IF st_config.b_config_fertig THEN
	(* Fehlermeldungen und Betriebsmeldungen ab dem Startindex in die globalen Meldungsarrays schreiben *)
	garr_stoermeldungen[st_config.i16_meld_startindex + 0] := sm_haspel_notaus;
	garr_stoermeldungen[st_config.i16_meld_startindex + 1] := sm_haspel_notabschaltung;
	garr_stoermeldungen[st_config.i16_meld_startindex + 2] := FALSE;
	garr_stoermeldungen[st_config.i16_meld_startindex + 3] := FALSE;
	garr_stoermeldungen[st_config.i16_meld_startindex + 4] := FALSE;
	garr_stoermeldungen[st_config.i16_meld_startindex + 5] := FALSE;
	garr_stoermeldungen[st_config.i16_meld_startindex + 6] := FALSE;
	garr_stoermeldungen[st_config.i16_meld_startindex + 7] := FALSE;
	garr_stoermeldungen[st_config.i16_meld_startindex + 8] := FALSE;
	garr_stoermeldungen[st_config.i16_meld_startindex + 9] := FALSE;
	garr_stoermeldungen[st_config.i16_meld_startindex + 10] := FALSE;
	garr_stoermeldungen[st_config.i16_meld_startindex + 11] := FALSE;
	garr_stoermeldungen[st_config.i16_meld_startindex + 12] := FALSE;
	garr_stoermeldungen[st_config.i16_meld_startindex + 13] := FALSE;
	garr_stoermeldungen[st_config.i16_meld_startindex + 14] := FALSE;
	garr_stoermeldungen[st_config.i16_meld_startindex + 15] := FALSE;
	garr_stoermeldungen[st_config.i16_meld_startindex + 16] := FALSE;
	garr_stoermeldungen[st_config.i16_meld_startindex + 17] := FALSE;
	garr_stoermeldungen[st_config.i16_meld_startindex + 18] := FALSE;
	garr_stoermeldungen[st_config.i16_meld_startindex + 19] := FALSE;
	
	garr_betriebsmeldungen[st_config.i16_meld_startindex + 0] := bm_haspel_bandende;
	garr_betriebsmeldungen[st_config.i16_meld_startindex + 1] := FALSE;
	garr_betriebsmeldungen[st_config.i16_meld_startindex + 2] := FALSE;
	garr_betriebsmeldungen[st_config.i16_meld_startindex + 3] := FALSE;
	garr_betriebsmeldungen[st_config.i16_meld_startindex + 4] := FALSE;
	garr_betriebsmeldungen[st_config.i16_meld_startindex + 5] := FALSE;
	garr_betriebsmeldungen[st_config.i16_meld_startindex + 6] := FALSE;
	garr_betriebsmeldungen[st_config.i16_meld_startindex + 7] := FALSE;
	garr_betriebsmeldungen[st_config.i16_meld_startindex + 8] := FALSE;
	garr_betriebsmeldungen[st_config.i16_meld_startindex + 9] := FALSE;
	garr_betriebsmeldungen[st_config.i16_meld_startindex + 10] := FALSE;
	garr_betriebsmeldungen[st_config.i16_meld_startindex + 11] := FALSE;
	garr_betriebsmeldungen[st_config.i16_meld_startindex + 12] := FALSE;
	garr_betriebsmeldungen[st_config.i16_meld_startindex + 13] := FALSE;
	garr_betriebsmeldungen[st_config.i16_meld_startindex + 14] := FALSE;
	garr_betriebsmeldungen[st_config.i16_meld_startindex + 15] := FALSE;
	garr_betriebsmeldungen[st_config.i16_meld_startindex + 16] := FALSE;
	garr_betriebsmeldungen[st_config.i16_meld_startindex + 17] := FALSE;
	garr_betriebsmeldungen[st_config.i16_meld_startindex + 18] := FALSE;
	garr_betriebsmeldungen[st_config.i16_meld_startindex + 19] := FALSE;
END_IF
END_FUNCTION_BLOCK

(* POU EPT Lib/CamEditor/ST_Kurvenscheibeneditor, ST *)
FUNCTION_BLOCK ST_Kurvenscheibeneditor
VAR_INPUT
 	udint_camtable_id						: UDINT;
	i16_laenge_mfp_tabelle				: UINT;
	arr_db_mfps							: ARRAY[1..ui_MAX_NUM_MFP] OF struct_db_motionfunctionpoint;	(* Vorgabe aus der Datenbank *)
	st_config								: struct_config;
	st_ctrl_in								: struct_ctrl_in;
END_VAR
VAR_IN_OUT
	i16_auftrag							: enum_auftrag_cameditor;
END_VAR
VAR_OUTPUT
	st_ctrl_out							: struct_ctrl_out;
END_VAR
VAR
	mc_point_id							: MC_MotionFunctionPoint_ID;
	mc_read_motion_function_point			: MC_ReadMotionFunctionPoint;
	mc_write_motion_function_point			: MC_WriteMotionFunctionPoint;
	arr_motion_function_points				: ARRAY[1..ui_MAX_NUM_MFP] OF MC_MotionFunctionPoint;	(* Eingelesene Kurvenscheibentabelle aus dem Systemmanager oder geschriebene MFPs an den Systemmanager *)
	udint_write_error_id 					: UDINT := 0;
	udint_read_error_id					: UDINT := 0;
	fb_state_entry							: ST_StateEntry;
	fb_ton_quitt							: TON;
	fb_ton_wz							: TON;
	fb_r_trig_ibn_lesen					: R_TRIG;
	fb_r_trig_ibn_schreiben					: R_TRIG;
	fb_ton_ibn_lesen						: TON;
	fb_ton_ibn_schreiben					: TON;
	b_ibn_lesen							: BOOL := FALSE;
	b_ibn_schreiben						: BOOL := FALSE;
	sm_fehler_schreibe_mfp 				: BOOL := FALSE;
	sm_fehler_lese_mfp					: BOOL := FALSE;
END_VAR
VAR CONSTANT
	ui_MAX_NUM_MFP					:UINT := 100;
END_VAR
fb_ton_wz(IN:= , PT:= , Q=> , ET=> );
fb_ton_quitt(IN:= , PT:= t#100ms, Q=> , ET=> );

fb_r_trig_ibn_lesen(CLK:= b_ibn_lesen, Q=> );
fb_r_trig_ibn_schreiben(CLK:= b_ibn_schreiben, Q=> );
fb_ton_ibn_lesen(IN:= , PT:= t#1s, Q=> , ET=> );
fb_ton_ibn_schreiben(IN:= , PT:= t#1s, Q=> , ET=> );


IF fb_r_trig_ibn_lesen.Q THEN
	fb_ton_ibn_lesen.IN := TRUE;
ELSE
	IF fb_ton_ibn_lesen.Q THEN
		b_ibn_lesen := FALSE;
	 	fb_ton_ibn_lesen.IN := FALSE;
	END_IF
END_IF

IF fb_r_trig_ibn_schreiben.Q THEN
	fb_ton_ibn_schreiben.IN := TRUE;
ELSE
	IF fb_ton_ibn_schreiben.Q THEN
		b_ibn_schreiben := FALSE;
	 	fb_ton_ibn_schreiben.IN := FALSE;
	END_IF
END_IF

(* ======================================Schrittkette======================================== *)
fb_state_entry(
	i16_next_step:= ,
	i16_pos:= 1,
	s_debugtext:= ,
	E=> ,
	X=> ,
	i16_step=> ,
	i16_last_step=> );

CASE fb_state_entry.i16_step OF
(*=======================================================*)
	0:	(* Init *)
		fb_ton_quitt.IN := FALSE;
		st_ctrl_out.b_bereit := FALSE;
		st_ctrl_out.b_fehler := FALSE;
		i16_auftrag := MFP_KEIN_AUFTRAG;
		mc_point_id := 1;
		mc_read_motion_function_point.Execute := FALSE;
		mc_write_motion_function_point.Execute := FALSE;
		sm_fehler_schreibe_mfp := FALSE;
		sm_fehler_lese_mfp := FALSE;
		fb_state_entry.i16_next_step := 10;

(*=======================================================*)
	10: (* Warte auf Auftrag *)
		IF fb_state_entry.E THEN
			st_ctrl_out.b_bereit := TRUE;
		END_IF

		(* Motion Function Points aus der Kurvenscheibentabelle des Systemmanagers lesen *)
		IF i16_auftrag = MFP_LESEN OR fb_r_trig_ibn_lesen.Q THEN
			fb_state_entry.i16_next_step := 100;
		(* Motion Function Points von der Datenbankvorgabe in die Kurvenscheibentabelle des Systemmanagers schreiben *)
		ELSIF i16_auftrag = MFP_SCHREIBEN OR fb_r_trig_ibn_schreiben.Q THEN
			fb_state_entry.i16_next_step := 200;
		END_IF

(*=======================================================*)
	100:
		mc_point_id := 1;
		fb_state_entry.i16_next_step := 110;

(*=======================================================*)
	110:	(* Lese die einzelnen MFPs aus der Kurvenscheibentabelle des Systemmanagers *)
		IF fb_state_entry.E THEN
			mc_read_motion_function_point.Execute := TRUE;
		END_IF

		IF mc_read_motion_function_point.Busy THEN
			mc_read_motion_function_point.Execute := FALSE;
			fb_state_entry.i16_next_step := 120;
		END_IF

(*=======================================================*)
	120:	(* MFP wurde gelesen *)
		IF  NOT mc_read_motion_function_point.Busy THEN
			IF NOT mc_read_motion_function_point.Error THEN
				fb_state_entry.i16_next_step := 130;
			ELSE
				sm_fehler_schreibe_mfp := TRUE;
				fb_state_entry.i16_next_step := FEHLER;
			END_IF
		END_IF

(*=======================================================*)
	130:	(* Zum nächsten MFP *)
		IF fb_state_entry.E THEN
			mc_point_id := mc_point_id + 1;
		END_IF

		IF mc_point_id > i16_laenge_mfp_tabelle THEN
			(* Alle Punkte wurden gelesen *)
			fb_state_entry.i16_next_step := 140;
		ELSE
			(* Weitere Punkte lesen *)
			fb_state_entry.i16_next_step := 110;
		END_IF

(*=======================================================*)
	140:	(* Lesevorgang beendet *)
		fb_state_entry.i16_next_step := 0;

(*=======================================================*)
	200:	(* Einlesen der Vorgabepunktetabelle *)
		IF fb_state_entry.E THEN
			FOR mc_point_id := 1  TO 32 BY 1DO
				arr_motion_function_points[mc_point_id].PointIndex := arr_db_mfps[mc_point_id].PointIndex;
				arr_motion_function_points[mc_point_id].FunctionType := arr_db_mfps[mc_point_id].FunctionType;
				arr_motion_function_points[mc_point_id].PointType := arr_db_mfps[mc_point_id].PointType;
				arr_motion_function_points[mc_point_id].RelIndexNextPoint := 1;
				arr_motion_function_points[mc_point_id].MasterPos := arr_db_mfps[mc_point_id].MasterPos;
				arr_motion_function_points[mc_point_id].SlavePos := arr_db_mfps[mc_point_id].SlavePos;
			END_FOR
		END_IF
		mc_point_id := 1;
		fb_state_entry.i16_next_step := 210;

(*=======================================================*)
	210:	(* Schreibe die einzelnen MFPs *)
		IF fb_state_entry.E THEN
			mc_write_motion_function_point.Execute := TRUE;
		END_IF

		IF mc_write_motion_function_point.Busy THEN
			mc_write_motion_function_point.Execute := FALSE;
			fb_state_entry.i16_next_step := 220;
		END_IF

(*=======================================================*)
	220:	(* MFP wurde geschrieben *)
		IF  NOT mc_write_motion_function_point.Busy THEN
			IF NOT  mc_write_motion_function_point.Error THEN
				fb_state_entry.i16_next_step := 230;
			ELSE
				sm_fehler_schreibe_mfp := TRUE;
				fb_state_entry.i16_next_step := FEHLER;
			END_IF
		END_IF

(*=======================================================*)
	230:	(* Zum nächsten MFP *)
		IF fb_state_entry.E THEN
			mc_point_id := mc_point_id + 1;
		END_IF

		IF mc_point_id > i16_laenge_mfp_tabelle THEN
			(* Alle Punkte wurden gelesen *)
			fb_state_entry.i16_next_step := 240;
		ELSE
			(* Weitere Punkte lesen *)
			fb_state_entry.i16_next_step := 210;
		END_IF

(*=======================================================*)
	240:	(* Schreibevorgang beendet *)
		fb_state_entry.i16_next_step := 0;

(*=======================================================*)
	1000: (* Fehler *)
		IF fb_state_entry.E THEN
			st_ctrl_out.b_fehler := TRUE;
			fb_ton_quitt.IN := FALSE;
		END_IF

		(*-----------------------Weiterschaltbedingungen----------------------------*)
		IF st_ctrl_in.b_quitt AND NOT fb_state_entry.E THEN
			st_ctrl_out.b_fehler := FALSE;
			fb_ton_quitt.IN := TRUE;
		END_IF

		IF fb_ton_quitt.Q THEN
			fb_ton_quitt.IN := FALSE;
			fb_state_entry.i16_next_step := 0;
		END_IF
END_CASE

fb_state_entry(
	i16_next_step:= ,
	i16_pos:= 2,
	s_debugtext:= ,
	E=> ,
	X=> ,
	i16_step=> ,
	i16_last_step=> );

mc_read_motion_function_point(
	Execute:= ,
	CamTableID:= udint_camtable_id,
	PointID:= mc_point_id,
	Point:= arr_motion_function_points[mc_point_id],
	Done=> , 
	Busy=> , 
	Error=> , 
	ErrorID=> );

mc_write_motion_function_point(
	Execute:= , 
	CamTableID:= udint_camtable_id,
	PointID:= mc_point_id,
	Point:= arr_motion_function_points[mc_point_id],
	Done=> , 
	Busy=> , 
	Error=> , 
	ErrorID=> );

IF st_config.b_config_fertig THEN
	garr_stoermeldungen[st_config.i16_meld_startindex + 0] := sm_fehler_lese_mfp;
	garr_stoermeldungen[st_config.i16_meld_startindex + 1] := sm_fehler_schreibe_mfp;
	garr_stoermeldungen[st_config.i16_meld_startindex + 2] := FALSE;
	garr_stoermeldungen[st_config.i16_meld_startindex + 3] := FALSE;
	garr_stoermeldungen[st_config.i16_meld_startindex + 4] := FALSE;
	garr_stoermeldungen[st_config.i16_meld_startindex + 5] := FALSE;
	garr_stoermeldungen[st_config.i16_meld_startindex + 6] := FALSE;
	garr_stoermeldungen[st_config.i16_meld_startindex + 7] := FALSE;
	garr_stoermeldungen[st_config.i16_meld_startindex + 8] := FALSE;
	garr_stoermeldungen[st_config.i16_meld_startindex + 9] := FALSE;
	garr_stoermeldungen[st_config.i16_meld_startindex + 10] := FALSE;
	garr_stoermeldungen[st_config.i16_meld_startindex + 11] := FALSE;
	garr_stoermeldungen[st_config.i16_meld_startindex + 12] := FALSE;
	garr_stoermeldungen[st_config.i16_meld_startindex + 13] := FALSE;
	garr_stoermeldungen[st_config.i16_meld_startindex + 14] := FALSE;
	garr_stoermeldungen[st_config.i16_meld_startindex + 15] := FALSE;
	garr_stoermeldungen[st_config.i16_meld_startindex + 16] := FALSE;
	garr_stoermeldungen[st_config.i16_meld_startindex + 17] := FALSE;
	garr_stoermeldungen[st_config.i16_meld_startindex + 18] := FALSE;
	garr_stoermeldungen[st_config.i16_meld_startindex + 19] := FALSE;
	
	garr_betriebsmeldungen[st_config.i16_meld_startindex + 0] := FALSE;
	garr_betriebsmeldungen[st_config.i16_meld_startindex + 1] := FALSE;
	garr_betriebsmeldungen[st_config.i16_meld_startindex + 2] := FALSE;
	garr_betriebsmeldungen[st_config.i16_meld_startindex + 3] := FALSE;
	garr_betriebsmeldungen[st_config.i16_meld_startindex + 4] := FALSE;
	garr_betriebsmeldungen[st_config.i16_meld_startindex + 5] := FALSE;
	garr_betriebsmeldungen[st_config.i16_meld_startindex + 6] := FALSE;
	garr_betriebsmeldungen[st_config.i16_meld_startindex + 7] := FALSE;
	garr_betriebsmeldungen[st_config.i16_meld_startindex + 8] := FALSE;
	garr_betriebsmeldungen[st_config.i16_meld_startindex + 9] := FALSE;
	garr_betriebsmeldungen[st_config.i16_meld_startindex + 10] := FALSE;
	garr_betriebsmeldungen[st_config.i16_meld_startindex + 11] := FALSE;
	garr_betriebsmeldungen[st_config.i16_meld_startindex + 12] := FALSE;
	garr_betriebsmeldungen[st_config.i16_meld_startindex + 13] := FALSE;
	garr_betriebsmeldungen[st_config.i16_meld_startindex + 14] := FALSE;
	garr_betriebsmeldungen[st_config.i16_meld_startindex + 15] := FALSE;
	garr_betriebsmeldungen[st_config.i16_meld_startindex + 16] := FALSE;
	garr_betriebsmeldungen[st_config.i16_meld_startindex + 17] := FALSE;
	garr_betriebsmeldungen[st_config.i16_meld_startindex + 18] := FALSE;
	garr_betriebsmeldungen[st_config.i16_meld_startindex + 19] := FALSE;
END_IF
END_FUNCTION_BLOCK

(* POU EPT Lib/CamEditor/Verfahrberechnungen/ST_MFCalcConstPhase, ST *)
FUNCTION_BLOCK ST_MFCalcConstPhase
VAR_INPUT
	st_config								: struct_config;
	st_ctrl_in								: struct_ctrl_in;

	(* Kurvenscheibendaten *)
	udiTableId							: MC_CAM_ID;			(* Table-ID *)
	eMotionFunctionType					: MC_MotionFunctionType;	(*Bewegungsgesetz: MOTIONFUNCTYPE_POLYNOM5 etc.*)
	i16_startpunkt_edit_mf_tab				: INT;
	arr_db_mf_tab						: ARRAY[1..i_MAX_NUM_MFP] OF struct_db_motionfunctionpoint;	(* Vorgabe aus der Datenbank *)

	(* Bewegungsdaten an der Last *)
	lrVeloMax							: LREAL;	(*maximale Geschwindigkeit [mm/s] an der Last *)
	lrAccMax								: LREAL;	(*maximale Beschleunigung [mm/s²] an der Last *)
	lrDecMax							: LREAL;	(*maximale Beschleunigung [mm/s²] an der Last *)

	lrModuloValue 						: LREAL ;
END_VAR
VAR_IN_OUT
	st_AxisRefMaster						: AXIS_REF;
	st_AxisRefSlave						: AXIS_REF;
END_VAR
VAR_OUTPUT
	lrMasterVeloMax						: LREAL;	(* Maximum Master Velocity [°/s] *)
	lrMasterRotPerMinMax					: LREAL;	(* Maximum Master Rotations per Minute [1/min] *)
	st_ctrl_out							: struct_ctrl_out;
END_VAR
VAR
	st_sm						 		: struct_cameditor_meldungen;
	fb_state_entry							: ST_StateEntry;
	fb_ton_quitt							: TON;
	fb_ton_wz							: TON;

	stMotionFunctionPointDummy			: MC_MotionFunctionPoint;	(* Dummy-Punkt *)
(*	TYPE MC_MotionFunctionPoint :
		STRUCT
		    PointIndex        		: MC_MotionFunctionPoint_ID;
		    FunctionType   		: MC_MotionFunctionType;
		    PointType         		: MC_MotionPointType;
		    RelIndexNextPoint 	: MC_MotionFunctionPoint_ID;
		    MasterPos         		: LREAL; (* X *)
		    SlavePos          		: LREAL; (* Y *)
		    SlaveVelo         		: LREAL; (* Y' *)
		    SlaveAcc          		: LREAL; (* Y'' *)
		    SlaveJerk         		: LREAL; (* Y''' *)
		END_STRUCT
	END_TYPE
*)

	(*Motion Function runterschreiben an NC*)
	astWriteMotionFunction 				: ARRAY[1..i_MAX_NUM_MFP] OF MC_MotionFunctionPoint;
	stWriteMFCamTableRef				: MC_CAM_Ref;	(*Definition Zieltabelle*)
	fbCamTableSelect					: MC_CamTableSelect;
	fbWriteMF							: MC_WriteMotionFunction;
	b_cam_table_select_periodic			: BOOL := FALSE;
	b_cam_table_select_master_absolute	: BOOL := FALSE;
	b_cam_table_select_slave_absolute		: BOOL := FALSE;

	(*Motion Function hochladen von NC*)
	fbReadMF							: MC_ReadMotionFunction;
	stReadMFCamTableRef				: MC_CAM_Ref;	(*Definition Zieltabelle*)
	astReadMotionFunction 				: ARRAY[0..i_MAX_NUM_MFP] OF MC_MotionFunctionPoint;

	(*Berechnung Konstantfahrphase*)
	fbMFcalcConstVelo					: ST_MFcalcConstVelo;	(*Baustein zur Berechnung, ob eine Konstantfahphase möglich ist*)
	stDataCalcConstVelo 					: ARRAY[1..4] OF MC_MotionFunctionPoint;	(*Aus der Berechnung ermittelte Punktedaten*)

	(* Berechnung Mastergeschwindigkeit*)
	fbMFMaxMasterVelo					: ST_MFMaxMasterVelo;	(* Baustein zur Berechnung der maximalen Mastergeschwindigkeit *)

	(*Temporäre Variablen *)
	iPointCount							: INT := 0;
	iNumMfPoints							: INT := 0;
	i_point_nr							: INT := 0;
	err_id								: UDINT := 0;
	i16_anzahl_mfps						: INT;
	lrStartPointMaster						: LREAL;	(* Startpunkt Master [°] *)
	lrStartPointSlave						: LREAL;	(* Startpunkt Slave [mm] *)
	lrEndPointMaster						: LREAL;	(* Endpunkt Master [°] *)
	lrEndPointSlave						: LREAL;	(* Endpunkt Slave [mm] *)
	lr_anfang_cam_table					: LREAL := 0;	(* Anfang Darstellungsbereich MF-Tabelle *)
	lr_ende_cam_table					: LREAL := 0;	(* Ende Darstellungsbereich MF-Tabelle *)
END_VAR
VAR CONSTANT
	i_MAX_NUM_MFP						: INT := 100;
END_VAR
fb_ton_wz(IN:= , PT:= , Q=> , ET=> );
fb_ton_quitt(IN:= , PT:= t#50ms, Q=> , ET=> );

(* ======================================Schrittkette======================================== *)
fb_state_entry(
	i16_next_step:= ,
	i16_pos:= 1,
	s_debugtext:= ,
	E=> ,
	X=> ,
	i16_step=> ,
	i16_last_step=> );

CASE fb_state_entry.i16_step OF
(*=======================================================*)
	0:	(* Init *)
		st_ctrl_out.b_bereit := FALSE;
		st_ctrl_out.b_fertig := FALSE;
		st_ctrl_out.b_fehler := FALSE;
		fbCamTableSelect.Execute := FALSE;
		fbWriteMF.Execute := FALSE;
		fbReadMF.Execute := FALSE;
		fbMFMaxMasterVelo.bExecute := FALSE;
		fbMFcalcConstVelo.bExecute := FALSE;
		err_id := 0;
		i16_anzahl_mfps := 0;
		st_sm.berechne_konstantfahrphase := FALSE;
		st_sm.berechne_max_master_geschwindigkeit := FALSE;
		st_sm.lese_camtable := FALSE;
		st_sm.lese_mfp := FALSE;
		st_sm.lesen_werte_mf_tab := FALSE;
		st_sm.schreibe_camtable := FALSE;
		st_sm.schreibe_mfp := FALSE;

		fb_state_entry.i16_next_step := 10;

(*=======================================================*)
	10:	(* Warte auf Start *)
		IF lrModuloValue > 0 THEN
			b_cam_table_select_periodic := TRUE;
			b_cam_table_select_master_absolute := TRUE;
			b_cam_table_select_slave_absolute := FALSE;
		ELSE
			b_cam_table_select_periodic := FALSE;
			b_cam_table_select_master_absolute := TRUE;
			b_cam_table_select_slave_absolute := TRUE;
		END_IF

		(*-----------------------Weiterschaltbedingungen----------------------------*)
		IF st_ctrl_in.b_start THEN
			i16_anzahl_mfps := 0;
			lrMasterVeloMax := 0;
			lrMasterRotPerMinMax := 0;
			fb_state_entry.i16_next_step := 100;
		END_IF

(*=======================================================*)
	100:	(*  *)
		IF fb_state_entry.E THEN
			FOR i_point_nr := 1 TO i_MAX_NUM_MFP BY 1 DO
				(*Für Download: Initialisieren aller  MFPs im Array *)
				astWriteMotionFunction[i_point_nr] := stMotionFunctionPointDummy;
				astWriteMotionFunction[i_point_nr].RelIndexNextPoint  := 1;

				(* Übernahme der Daten aus der WKZ-Datenbank *)
				astWriteMotionFunction[i_point_nr].FunctionType := arr_db_mf_tab[i_point_nr].FunctionType;
				astWriteMotionFunction[i_point_nr].MasterPos  := arr_db_mf_tab[i_point_nr].MasterPos;
				astWriteMotionFunction[i_point_nr].SlavePos  := arr_db_mf_tab[i_point_nr].SlavePos;
				astWriteMotionFunction[i_point_nr].PointType  := arr_db_mf_tab[i_point_nr].PointType;
				astWriteMotionFunction[i_point_nr].PointIndex  := arr_db_mf_tab[i_point_nr].PointIndex;

				IF astWriteMotionFunction[i_point_nr].FunctionType > MOTIONFUNCTYPE_NOTDEF THEN
					i16_anzahl_mfps := i16_anzahl_mfps + 1;
				END_IF
			END_FOR

			(* Beim Letzen Punkt in der Tabelle immer den RelIndexNextPoint auf 0 setzen *)
			astWriteMotionFunction[i16_anzahl_mfps].RelIndexNextPoint := 0;

			(* Darstellungsbereich der MF-Tabelle (wird benötigt für die Funktion "MC_ReadMotionFunctionValues") *)
			IF lrModuloValue > 0 THEN
				lr_anfang_cam_table := 0;
				lr_ende_cam_table := lrModuloValue;
			ELSE
				lr_anfang_cam_table := arr_db_mf_tab[1].MasterPos;
				lr_ende_cam_table := arr_db_mf_tab[i16_anzahl_mfps].MasterPos;
			END_IF
		END_IF

		(*-----------------------Weiterschaltbedingungen----------------------------*)
		fb_state_entry.i16_next_step := 110;


(*=======================================================*)
	110:	(* Starte Berechnung der Konstantfahrphase *)
		IF fb_state_entry.E THEN
			fbMFcalcConstVelo.bExecute := TRUE;
		END_IF

		(*-----------------------Weiterschaltbedingungen----------------------------*)
		IF fbMFcalcConstVelo.bBusy THEN
			fb_state_entry.i16_next_step := 120;
		END_IF

(*=======================================================*)
	120:	(* Starte Berechnung der Konstantfahrphase *)
		IF NOT fbMFcalcConstVelo.bBusy THEN
			IF fbMFcalcConstVelo.bDone THEN
				fbMFcalcConstVelo.bExecute := FALSE;
				IF fbMFcalcConstVelo.bConstantVelo THEN
					iNumMfPoints := i16_anzahl_mfps + 2;
					fb_state_entry.i16_next_step := 130;
				ELSE
					iNumMfPoints := i16_anzahl_mfps;
					fb_state_entry.i16_next_step := 140;
				END_IF
			ELSIF fbMFcalcConstVelo.bError THEN
				st_sm.berechne_konstantfahrphase := TRUE;
				fb_state_entry.i16_next_step := 1000;
			END_IF
		END_IF

(*=======================================================*)
	130:	(* Auswertung ob Konstantfahrphase *)
		IF fb_state_entry.E THEN
			(* Verschieben aller weiteren Punkte um 2 Positionen nach hinten *)
			FOR i_point_nr := iNumMfPoints TO (i16_startpunkt_edit_mf_tab + 1) BY -1 DO
				astWriteMotionFunction[i_point_nr] := astWriteMotionFunction[i_point_nr - 2];
				astWriteMotionFunction[i_point_nr].PointIndex := i_point_nr;
			END_FOR

			iPointCount := i16_startpunkt_edit_mf_tab;

			(*Startpunkt: spezifische Daten anpassen*)
			astWriteMotionFunction[iPointCount].MasterPos := stDataCalcConstVelo[1].MasterPos;
			astWriteMotionFunction[iPointCount].SlavePos := stDataCalcConstVelo[1].SlavePos;
			astWriteMotionFunction[iPointCount].SlaveVelo := stDataCalcConstVelo[1].SlaveVelo;
			astWriteMotionFunction[iPointCount].SlaveJerk := stDataCalcConstVelo[1].SlaveJerk;
			(*Punktetyp eintragen*)
			astWriteMotionFunction[iPointCount].RelIndexNextPoint := 1;
			astWriteMotionFunction[iPointCount].FunctionType := stDataCalcConstVelo[1].FunctionType;
			astWriteMotionFunction[iPointCount].PointIndex := iPointCount;
			astWriteMotionFunction[iPointCount].PointType := stDataCalcConstVelo[1].PointType;

			iPointCount := iPointCount + 1;

			(*Zwischenpunkt 1: Konstantfahrphase eintragen*)
			astWriteMotionFunction[iPointCount].MasterPos := stDataCalcConstVelo[2].MasterPos;
			astWriteMotionFunction[iPointCount].SlavePos := stDataCalcConstVelo[2].SlavePos;
			astWriteMotionFunction[iPointCount].SlaveVelo := stDataCalcConstVelo[2].SlaveVelo;
			astWriteMotionFunction[iPointCount].SlaveJerk := stDataCalcConstVelo[2].SlaveJerk;
			(*Punktetyp eintragen*)
			astWriteMotionFunction[iPointCount].RelIndexNextPoint := 1;
			astWriteMotionFunction[iPointCount].FunctionType := stDataCalcConstVelo[2].FunctionType;
			astWriteMotionFunction[iPointCount].PointIndex := iPointCount;
			astWriteMotionFunction[iPointCount].PointType := stDataCalcConstVelo[2].PointType;
	
			iPointCount := iPointCount + 1;
	
			(*Zwischenpunkt 2: Konstantfahrphase eintragen*)
			astWriteMotionFunction[iPointCount].MasterPos := stDataCalcConstVelo[3].MasterPos;
			astWriteMotionFunction[iPointCount].SlavePos := stDataCalcConstVelo[3].SlavePos;
			astWriteMotionFunction[iPointCount].SlaveVelo := stDataCalcConstVelo[3].SlaveVelo;
			astWriteMotionFunction[iPointCount].SlaveJerk := stDataCalcConstVelo[3].SlaveJerk;
			(*Punktetyp eintragen*)
			astWriteMotionFunction[iPointCount].RelIndexNextPoint := 1;
			astWriteMotionFunction[iPointCount].FunctionType := stDataCalcConstVelo[3].FunctionType;
			astWriteMotionFunction[iPointCount].PointIndex := iPointCount;
			astWriteMotionFunction[iPointCount].PointType := stDataCalcConstVelo[3].PointType;

			iPointCount := iPointCount + 1;

			(* Beim Letzen Punkt in der Tabelle immer den RelIndexNextPoint auf 0 setzen *)
			astWriteMotionFunction[i16_anzahl_mfps + 2].RelIndexNextPoint := 0;
		END_IF

		(*-----------------------Weiterschaltbedingungen----------------------------*)
		fb_state_entry.i16_next_step := 140;

(*=======================================================*)
	140:	(* Alle Punkte der MF-Tabelle werden an die NC runter geschrieben  *)
		IF fb_state_entry.E THEN
			(*Tabelle initialisieren *)
			stWriteMFCamTableRef.pArray := ADR(astWriteMotionFunction[1]);	(* Adresse des ersten eindimensionalen Arrays vom Typ MC_MotionFunctionPoint. Jedes Array-Element enthält eine Beschreibung einer Stützstelle der Kurvenscheibe. *)
			stWriteMFCamTableRef.ArraySize := SIZEOF(astWriteMotionFunction[1]) * iNumMfPoints;
			stWriteMFCamTableRef.TableType := MC_TABLETYPE_MOTIONFUNCTION;
			stWriteMFCamTableRef.NoOfColumns := 1;	(* Bei Table Type "MC_TABLETYPE_MOTIONFUNCTION" ist NoOfColumns immer 1 *)
			stWriteMFCamTableRef.NoOfRows := iNumMfPoints;

			fbCamTableSelect.Execute := TRUE;
		END_IF

		(*-----------------------Weiterschaltbedingungen----------------------------*)
		IF fbCamTableSelect.Busy THEN
			fb_state_entry.i16_next_step := 150;
		END_IF

(*=======================================================*)
	150:	(* Alle Punkte der MF-Tabelle werden an die NC runter geschrieben  *)
		IF NOT fbCamTableSelect.Busy THEN
			IF fbCamTableSelect.Done THEN
				fbCamTableSelect.Execute := FALSE;
				fb_state_entry.i16_next_step := 200;
			ELSIF fbCamTableSelect.Error THEN
				st_sm.schreibe_camtable := TRUE;
				err_id := fbCamTableSelect.ErrorID;
				fb_state_entry.i16_next_step := 1000;
			END_IF
		END_IF

(*=======================================================*)
	200:	(* Lesen der MF-Tabelle von der NC  *)
		IF fb_state_entry.E THEN
			stReadMFCamTableRef.pArray := ADR(astReadMotionFunction[0]);
			stReadMFCamTableRef.ArraySize := SIZEOF(astReadMotionFunction[0]) * (iNumMfPoints + 1) ;
			stReadMFCamTableRef.NoOfColumns := 2;		(* Master und Slave Spalte*)
			stReadMFCamTableRef.NoOfRows := iNumMfPoints;
			stReadMFCamTableRef.TableType := MC_TABLETYPE_MOTIONFUNCTION;
			
			(* Für Upload initialisieren *)
			FOR iPointCount := 1 TO i_MAX_NUM_MFP DO
				astReadMotionFunction[iPointCount] := stMotionFunctionPointDummy;
			END_FOR

			fbReadMF.Execute := TRUE;
		END_IF

		(*-----------------------Weiterschaltbedingungen----------------------------*)
		IF fbReadMF.Busy THEN
			fb_state_entry.i16_next_step := 210;
		END_IF

(*=======================================================*)
	210:	(* Die gesamte MF-Tabelle hochladen  *)
		IF NOT fbReadMF.Busy THEN
			IF fbReadMF.Done THEN
				fbReadMF.Execute := FALSE;
				fb_state_entry.i16_next_step := 220;
			ELSIF fbReadMF.Error THEN
				st_sm.lese_camtable := TRUE;
				err_id := fbReadMF.ErrorID;
				fb_state_entry.i16_next_step := 1000;
			END_IF
		END_IF

(*=======================================================*)
	220:	(* Grenzhubzahlberechung  *)
		IF fb_state_entry.E THEN
			fbMFMaxMasterVelo.bExecute := TRUE;
		END_IF

		(*-----------------------Weiterschaltbedingungen----------------------------*)
		IF fbMFMaxMasterVelo.bBusy THEN
			fb_state_entry.i16_next_step := 230;
		END_IF

(*=======================================================*)
	230:	(* Berechnung fertig  *)
		IF NOT fbMFMaxMasterVelo.bBusy THEN
			IF fbMFMaxMasterVelo.bDone THEN
				fbMFMaxMasterVelo.bExecute := FALSE;
				fb_state_entry.i16_next_step := 240;
			ELSIF fbMFMaxMasterVelo.bError THEN
				st_sm.berechne_max_master_geschwindigkeit := TRUE;
				err_id := fbMFMaxMasterVelo.udiErrorId;
				fb_state_entry.i16_next_step := 1000;
			END_IF
		END_IF

(*=======================================================*)
	240:	(* Zuweisung der maximalen Mastergeschwindigkeit *)
		IF fb_state_entry.E THEN
			lrMasterVeloMax := fbMFMaxMasterVelo.lrMasterVeloMax;
			IF lrModuloValue > 0 THEN
				lrMasterRotPerMinMax := 60.0 * lrMasterVeloMax / lrModuloValue;
			ELSE
				lrMasterRotPerMinMax := 0;
			END_IF
		END_IF

		(*-----------------------Weiterschaltbedingungen----------------------------*)
		fb_state_entry.i16_next_step := 250;

(*=======================================================*)
	250:	(* Fertig  *)
		IF fb_state_entry.E THEN
			st_ctrl_out.b_fertig := TRUE;
		END_IF

		(*-----------------------Weiterschaltbedingungen----------------------------*)
		IF NOT st_ctrl_in.b_start THEN
			st_ctrl_out.b_fertig := FALSE;
			fb_state_entry.i16_next_step := 10;
		END_IF

(*=======================================================*)
	FEHLER: (* Fehler *)
		IF fb_state_entry.E THEN
			st_ctrl_out.b_fehler := TRUE;
			fb_ton_quitt.IN := FALSE;
		END_IF

		(*-----------------------Weiterschaltbedingungen----------------------------*)
		IF st_ctrl_in.b_quitt AND NOT fb_state_entry.E THEN
			st_ctrl_out.b_fehler := FALSE;
			fb_ton_quitt.IN := TRUE;
		END_IF

		IF fb_ton_quitt.Q THEN
			fb_ton_quitt.IN := FALSE;
			fb_state_entry.i16_next_step := 0;
		END_IF
END_CASE

fb_state_entry(
	i16_next_step:= ,
	i16_pos:= 2,
	s_debugtext:= ,
	E=> ,
	X=> ,
	i16_step=> ,
	i16_last_step=> );

(* Erstellen einer neuen MF-Tabelle mit anschliessendem Füllen der Punktdaten: *)
(* Es wird eine neue Tabelle in der NC angelegt zudem werden  Master und Slave Achsen zugeordnet. *)
(* Die Länge der Tabelle mit ihren Punktdaten wird gleichzeitig mit reingeschrieben. *)
fbCamTableSelect(
	Execute:= , 
	Periodic:= b_cam_table_select_periodic,
	MasterAbsolute:= b_cam_table_select_master_absolute,
	SlaveAbsolute:= b_cam_table_select_slave_absolute,
	CamTableID:= udiTableId,
	Master := st_AxisRefMaster,
	Slave := st_AxisRefSlave,
	CamTable:= stWriteMFCamTableRef,
	Done=> ,
	Busy=> , 
	Error=> , 
	ErrorID=> );

(* Die gesamte Tabelle einlesen aus der NC *)
fbReadMF(
	Execute:= ,
	CamTableID:= udiTableId,
	PointID:= 1,
	NumPoints:= stReadMFCamTableRef.NoOfRows,
	CamTable:= stReadMFCamTableRef,
	Done=> ,
	Busy=> ,
	Error=> ,
	ErrorID=> ,
	NumPointsRead=> );

(* Die ganze oder einen Teil der MF-Tabelle schreiben *)
fbWriteMF(
	Execute:= ,
	CamTableID:= udiTableId,
	PointID:= i16_startpunkt_edit_mf_tab,
	NumPoints:= i16_anzahl_mfps,
	CamTable:= stWriteMFCamTableRef,
	Done=> ,
	Busy=> , 
	Error=> , 
	ErrorID=> );

(* Berechnen ob Konstantfahrphase möglich *)
fbMFcalcConstVelo(
	bExecute:= ,
	eMotionFunctionType:= eMotionFunctionType,
	lrStartPointMaster:= arr_db_mf_tab[i16_startpunkt_edit_mf_tab].MasterPos,
	lrStartPointSlave:= arr_db_mf_tab[i16_startpunkt_edit_mf_tab].SlavePos,
	lrEndPointMaster:= arr_db_mf_tab[i16_startpunkt_edit_mf_tab + 1].MasterPos,
	lrEndPointSlave:= arr_db_mf_tab[i16_startpunkt_edit_mf_tab + 1].SlavePos,
	lrVeloLimit:= lrVeloMax,
	lrAccLimit:= lrAccMax,
	lrDecLimit:= lrDecMax,
	lrModuloValue:= lrModuloValue,
	stData:= stDataCalcConstVelo,
	bDone=> ,
	bError=> ,
	szErrText=> ,
	bConstantVelo=> ,
	lrVeloRef=> ,	(* Momentan nicht verwendet *)
	lrAccRef=> );	(* Momentan nicht verwendet *)

(* Berechne maximal mögliche Mastergeschwindigkeit *)
fbMFMaxMasterVelo(
	bExecute:= ,
	bEvCamTableChar:= eMotionFunctionType = MOTIONFUNCTYPE_POLYNOM7_MM,
	udiSlaveTableId:= udiTableId,
	lrVeloMax:= lrVeloMax,
	lrAccMax:= lrAccMax,
	lrDecMax:= lrDecMax,
	i16_anzahl_mfps:= iNumMfPoints,
	lr_anfang_cam_table:= lr_anfang_cam_table,
	lr_ende_cam_table:= lr_ende_cam_table,
	bDone=> ,
	bError=> , 
	udiErrorId=> ,
	szErrText=> ,
	lrMasterVeloMax=> );

IF st_config.b_config_fertig THEN
	garr_stoermeldungen[st_config.i16_meld_startindex + 0] := st_sm.lese_mfp;
	garr_stoermeldungen[st_config.i16_meld_startindex + 1] := st_sm.lese_camtable;
	garr_stoermeldungen[st_config.i16_meld_startindex + 2] := st_sm.lesen_werte_mf_tab;
	garr_stoermeldungen[st_config.i16_meld_startindex + 3] := st_sm.schreibe_mfp;
	garr_stoermeldungen[st_config.i16_meld_startindex + 4] := st_sm.schreibe_camtable;
	garr_stoermeldungen[st_config.i16_meld_startindex + 5] := st_sm.berechne_konstantfahrphase;
	garr_stoermeldungen[st_config.i16_meld_startindex + 6] := st_sm.berechne_max_master_geschwindigkeit;
	garr_stoermeldungen[st_config.i16_meld_startindex + 7] := FALSE;
	garr_stoermeldungen[st_config.i16_meld_startindex + 8] := FALSE;
	garr_stoermeldungen[st_config.i16_meld_startindex + 9] := FALSE;
	garr_stoermeldungen[st_config.i16_meld_startindex + 10] := FALSE;
	garr_stoermeldungen[st_config.i16_meld_startindex + 11] := FALSE;
	garr_stoermeldungen[st_config.i16_meld_startindex + 12] := FALSE;
	garr_stoermeldungen[st_config.i16_meld_startindex + 13] := FALSE;
	garr_stoermeldungen[st_config.i16_meld_startindex + 14] := FALSE;
	garr_stoermeldungen[st_config.i16_meld_startindex + 15] := FALSE;
	garr_stoermeldungen[st_config.i16_meld_startindex + 16] := FALSE;
	garr_stoermeldungen[st_config.i16_meld_startindex + 17] := FALSE;
	garr_stoermeldungen[st_config.i16_meld_startindex + 18] := FALSE;
	garr_stoermeldungen[st_config.i16_meld_startindex + 19] := FALSE;
	
	garr_betriebsmeldungen[st_config.i16_meld_startindex + 0] := FALSE;
	garr_betriebsmeldungen[st_config.i16_meld_startindex + 1] := FALSE;
	garr_betriebsmeldungen[st_config.i16_meld_startindex + 2] := FALSE;
	garr_betriebsmeldungen[st_config.i16_meld_startindex + 3] := FALSE;
	garr_betriebsmeldungen[st_config.i16_meld_startindex + 4] := FALSE;
	garr_betriebsmeldungen[st_config.i16_meld_startindex + 5] := FALSE;
	garr_betriebsmeldungen[st_config.i16_meld_startindex + 6] := FALSE;
	garr_betriebsmeldungen[st_config.i16_meld_startindex + 7] := FALSE;
	garr_betriebsmeldungen[st_config.i16_meld_startindex + 8] := FALSE;
	garr_betriebsmeldungen[st_config.i16_meld_startindex + 9] := FALSE;
	garr_betriebsmeldungen[st_config.i16_meld_startindex + 10] := FALSE;
	garr_betriebsmeldungen[st_config.i16_meld_startindex + 11] := FALSE;
	garr_betriebsmeldungen[st_config.i16_meld_startindex + 12] := FALSE;
	garr_betriebsmeldungen[st_config.i16_meld_startindex + 13] := FALSE;
	garr_betriebsmeldungen[st_config.i16_meld_startindex + 14] := FALSE;
	garr_betriebsmeldungen[st_config.i16_meld_startindex + 15] := FALSE;
	garr_betriebsmeldungen[st_config.i16_meld_startindex + 16] := FALSE;
	garr_betriebsmeldungen[st_config.i16_meld_startindex + 17] := FALSE;
	garr_betriebsmeldungen[st_config.i16_meld_startindex + 18] := FALSE;
	garr_betriebsmeldungen[st_config.i16_meld_startindex + 19] := FALSE;
END_IF
END_FUNCTION_BLOCK

(* POU EPT Lib/CamEditor/Verfahrberechnungen/ST_MFcalcConstVelo, ST *)
FUNCTION_BLOCK ST_MFcalcConstVelo
VAR_INPUT
	bExecute			: BOOL;
	eMotionFunctionType	: MC_MotionFunctionType;(*Bewegungsgesetz*)
	lrStartPointMaster		: LREAL;	(* Start Point Master [°] oder [mm] *)
	lrStartPointSlave		: LREAL;	(* Start Point Slave [mm] *)
	lrEndPointMaster		: LREAL;	(* End Point Master [°] oder [mm] *)
	lrEndPointSlave		: LREAL;	(* End Point Slave [mm] *)
	lrVeloLimit			: LREAL;	(*Slave Geschwindigkeitsgrenzwert [EINH/s]*)
	lrAccLimit			: LREAL;	(*Slave Beschleunigungsgrenzwert [EINH/s²]*)
	lrDecLimit			: LREAL;	(*Slave Bremsbeschleunigungsgrenzwert [EINH/s²]*)
	lrModuloValue		: LREAL;	(*Modulo-Periode des Master-Zyklus*)
END_VAR
VAR_OUTPUT
	bBusy				: BOOL;
	bDone 				: BOOL;
	bError 				: BOOL;

	bConstantVelo		: BOOL;	(* Ergebnis aus der Berechnung der Konstantfahrphase *)

	lrVeloRef			: LREAL;	(* referenced velocity *)
	lrAccRef				: LREAL;	(* referenced acceleration *)
END_VAR
VAR_IN_OUT
	stData 				: ARRAY[1..4] OF MC_MotionFunctionPoint; (*Berechnete Punktedaten*)
END_VAR
VAR
	szErrText			: STRING;		(*Error text*)
	lrVMax				: LREAL;			(*Slave Geschwindigkeit [m/s]*)
	lrAMax				: LREAL;			(*Slave Beschleunigung [m/s²]*)
	lrDMax				: LREAL;			(*Slave Verzögerung [m/s²] *)
	lrCvOrig				: LREAL;			(*Original Bewegungsgesetz*)
	lrCaOrig				: LREAL;			(*Original Bewegungsgesetz*)
	lrCv					: LREAL;			(*Polynom 5*)
	lrCa					: LREAL;			(*Polynom 5*)
	eMfType				: MC_MotionFunctionType;	(*Polynom 5*)
	lrPhiAcc				: LREAL;			(*Beschleunigungsphase*)
	lrPhiVelo				: LREAL;			(*Bewegungsphase v=const.*)
	lrPhi					: LREAL;			(*Gesamtbewegungsphase*)
	lrTAcc				: LREAL;			(*Beschleunigungszeit*)
	lrTVelo_to_TAcc		: LREAL;			(*Quotient Konstantfahrt / Beschleunigungsfahrt*)
	lrXAccOrig			: LREAL;			(*Original Beschleunigungsweg*)
	lrXAcc				: LREAL;			(*Beschleunigungsweg*)

	lrTDec				: LREAL;			(*Bremsszeit*)
	lrXDecOrig			: LREAL;			(*Original Bremssweg*)
	lrXDec				: LREAL;			(*Bremssweg*)

	lrXVelo				: LREAL;			(*Konstantfahrweg*)
	lrX					: LREAL;			(*Gesamtweg / Hub*)
	lrV					: LREAL;			(*Geschwindigkeit*)

	fb_state_entry			: ST_StateEntry;
END_VAR
(* ======================================Schrittkette======================================== *)
fb_state_entry(
	i16_next_step:= ,
	i16_pos:= 1,
	s_debugtext:= ,
	E=> ,
	X=> ,
	i16_step=> ,
	i16_last_step=> );

CASE fb_state_entry.i16_step OF
(*=======================================================*)
	0 :	(* Init*)
		bBusy := FALSE;
		bDone := FALSE;
		bError := FALSE;
		bConstantVelo := FALSE;
		szErrText := '';
		fb_state_entry.i16_next_step := 10;

(*=======================================================*)
	10:	(* Warte Execute *)

		(*-----------------------Weiterschaltbedingungen----------------------------*)
		IF bExecute THEN
			bBusy := TRUE;
			fb_state_entry.i16_next_step := 20;
		END_IF

(*=======================================================*)
	20:
		IF fb_state_entry.E THEN
			(* Die Variable lrPhi wird für lineare und runde(modulo) Master verwendet *)
 			IF lrModuloValue = 0 THEN
				(*Linearachse: Einheiten umrechnen*)
				lrX := lrEndPointSlave - lrStartPointSlave;
				lrPhi := ABS(lrEndPointMaster - lrStartPointMaster);
			ELSE
				(*Rundachse: Einheiten umrechnen*)
				lrX := lrEndPointSlave - lrStartPointSlave;
				lrPhi := MODABS(lrEndPointMaster - lrStartPointMaster, lrModuloValue);
				(* Sonderfall: phi4 - phi1 = modulowert *)
				IF (lrEndPointMaster - lrStartPointMaster = lrModuloValue) THEN
					lrPhi := lrModuloValue;
				END_IF
			END_IF

			lrVMax := lrVeloLimit;
			lrAMax := lrAccLimit;
			lrDMax := lrDecLimit;
			
			(*Bewegungsgesetz auswaehlen -> Charakteristische Werte Cv, Ca*)
			IF eMotionFunctionType = MOTIONFUNCTYPE_POLYNOM7_MM THEN
			(*Polynom 7*)
				lrCvOrig :=1.9;
				lrCaOrig :=7.51;
				eMfType := MOTIONFUNCTYPE_POLYNOM7_MM;
				lrCv :=1.9;
				lrCa :=7.51;
			
			ELSE
			(*Polynom 5*)
				lrCvOrig :=1.88;
				lrCaOrig :=5.78;
				eMfType := MOTIONFUNCTYPE_POLYNOM5_MM;
				lrCv :=1.88;
				lrCa :=5.78;
			END_IF

			(*Plausibilitaetsprüfung*)
			IF lrAMax <= 0 THEN
				fb_state_entry.i16_next_step := FEHLER;
				szErrText := 'Amax <= 0';
			ELSIF lrDMax <= 0 THEN
				fb_state_entry.i16_next_step := FEHLER;
				szErrText := 'Dmax <= 0';
			ELSIF lrVMax <= 0 THEN
				fb_state_entry.i16_next_step := FEHLER;
				szErrText := 'Vmax <= 0';
			ELSIF lrCv <= 0 THEN
				fb_state_entry.i16_next_step := FEHLER;
				szErrText := 'Cv <= 0';
			ELSIF lrCa <= 0 THEN
				fb_state_entry.i16_next_step := FEHLER;
				szErrText := 'Ca <= 0';
			ELSIF lrX = 0 THEN
				fb_state_entry.i16_next_step := FEHLER;
				szErrText := 'x = 0';
			ELSIF lrPhi <= 0 THEN
				fb_state_entry.i16_next_step := FEHLER;
				szErrText := 'phi <= 0';
			ELSE
				fb_state_entry.i16_next_step := 30;
			END_IF
		END_IF

(*=======================================================*)
	30:
		IF fb_state_entry.E THEN
			(*Berechnung: Weg, ab dem sich das Einfuegen einer Konstantfahrphase lohnt*)
			(*
			Bewegungsgesetzt der Translation: s = 0.5 * v * t = 0.5 * v^2 / a
			----------------------------------
			xAcc = 0.5 * (vmax² * Ca) / (Cv² * amax)
			xDec = 0.5 * (vmax² * Ca) / (Cv² * dmax)
			----------------------------------
			
			x		:	Gesamtweg (Hub)
			xAcc	:	Weg beim Fahren mit max. Beschleunigung, so dass die max. Geschwind. gerade erreicht wird
			xDec	:	Weg beim Fahren mit max. Verzögerung, so dass die max. Geschwind. gerade erreicht wird
			vmax	:	max. zulaessige Geschwindigkeit
			amax	:	max. zulaessige Beschleunigung
			dmax	:	max. zulaessige Verzoegerung
			Cv		:	Geschwindigkeitskennwert des Bewegungsgesetzes
			Ca		:	Beschleunigungskennwert des Bewegungsgesetzes
			*)
			
			lrXAcc := 0.5 * (lrVMax * lrVMax * lrCa) / (lrCv * lrCv * lrAMax);
			lrXAcc := F_rSign(lrX) * lrXAcc;
			lrXAccOrig := 0.5 * (lrVMax * lrVMax * lrCaOrig) / (lrCvOrig * lrCvOrig * lrAMax);
			
			lrXDec := 0.5 * (lrVMax * lrVMax * lrCa) / (lrCv * lrCv * lrDMax);
			lrXDec := F_rSign(lrX) * lrXDec;
			lrXDecOrig := 0.5 * (lrVMax * lrVMax * lrCaOrig) / (lrCvOrig * lrCvOrig * lrDMax);
			
			IF (lrXAccOrig + lrXDecOrig) < ABS(lrX) THEN
				bConstantVelo := TRUE;

				(*Berechnung Wertebereich fuer Beschleunigungsphase ohne Konstantfahrtanteil*)
				(*
				t = v / a
				--------------------------------
				tAcc = (vmax * Ca) / (Cv * amax)
				--------------------------------
				*)
				lrTAcc := (lrVMax * lrCa) / (lrAMax * lrCv);
				lrTDec := (lrVMax * lrCa) / (lrDMax * lrCv);
				(*
				---------------------------------------
				tVelo/tAcc = (x - xAcc) / (vmax * tAcc)
				---------------------------------------
				*)
				lrTVelo_to_TAcc := ABS(lrX - lrXAcc - lrXDec) / (lrVMax * (lrTAcc + lrTDec)/2);
				(*
				---------------------------------------
				tAcc = phi / {[(x - xAcc)/(vmax * tAcc)] + 1}
				---------------------------------------
				*)
				lrPhiAcc := lrPhi / (lrTVelo_to_TAcc + 1);
				lrPhiVelo := lrPhi - lrPhiAcc;

				lrXVelo := lrX - lrXAcc - lrXDec;
				lrV := lrXVelo / lrPhiVelo;

				(*Berechnete MFP Daten*)
				stData[1].FunctionType := eMfType;
				stData[1].PointType := MOTIONPOINTTYPE_VELOCITY;
				stData[1].MasterPos := lrStartPointMaster;
				stData[1].SlavePos := lrStartPointSlave;
				stData[1].SlaveVelo := lrV;
				
				stData[2].FunctionType := MOTIONFUNCTYPE_POLYNOM1;
				stData[2].PointType := MOTIONPOINTTYPE_VELOCITY;
				stData[2].MasterPos := lrStartPointMaster + (lrPhiAcc *  lrDecLimit / (lrAccLimit + lrDecLimit));
				stData[2].SlavePos := lrStartPointSlave + lrXAcc;
				stData[2].SlaveVelo := lrV;
				
				stData[3].FunctionType := eMfType;
				stData[3].PointType := MOTIONPOINTTYPE_VELOCITY;
				stData[3].MasterPos := lrEndPointMaster - (lrPhiAcc * lrAccLimit  / (lrAccLimit + lrDecLimit));
				stData[3].SlavePos := lrEndPointSlave - lrXDec;
				stData[3].SlaveVelo := lrV;
				
				stData[4].FunctionType := eMfType;
				stData[4].PointType := MOTIONPOINTTYPE_REST;
				stData[4].MasterPos := lrEndPointMaster;
				stData[4].SlavePos := lrEndPointSlave;
				stData[4].SlaveVelo := 0;
				
				lrVeloRef := ABS(lrV);
				lrAccRef := MAX(lrAccLimit,lrDecLimit) * (EXPT(lrVeloRef /lrVeloLimit,2));

			ELSE
				bConstantVelo := FALSE;
			END_IF
			fb_state_entry.i16_next_step := 40;
		END_IF

(*=======================================================*)
	40: (* Fertig *)
		IF fb_state_entry.E THEN
			bBusy := FALSE;
			bDone := TRUE;
		END_IF

		(*-----------------------Weiterschaltbedingungen----------------------------*)
		IF NOT bExecute AND NOT fb_state_entry.E THEN
			 bDone := FALSE;
			fb_state_entry.i16_next_step := 10;
		END_IF

(*=======================================================*)
	1000: (* Fehler *)
		IF fb_state_entry.E THEN
			bError := TRUE;
			bBusy := FALSE;
		END_IF

		(*-----------------------Weiterschaltbedingungen----------------------------*)
		IF NOT bExecute THEN
			fb_state_entry.i16_next_step := 0;
		END_IF
END_CASE

fb_state_entry(
	i16_next_step:= ,
	i16_pos:= 2,
	s_debugtext:= ,
	E=> ,
	X=> ,
	i16_step=> ,
	i16_last_step=> );
END_FUNCTION_BLOCK

(* POU EPT Lib/CamEditor/Verfahrberechnungen/ST_MFMaxMasterVelo, ST *)
FUNCTION_BLOCK ST_MFMaxMasterVelo
VAR_INPUT
	bExecute 						: BOOL;
	enu_mastertyp					: enum_ecd_typ;	(* Master ist Rund- oder Linearachse *)
	bEvCamTableChar				: BOOL;
	udiSlaveTableId					: MC_CAM_ID;	(* Slave Table-ID *)

	(* Bewegungsdaten Slave *)
	lrVeloMax						: LREAL;	(*maximale Geschwindigkeit [mm/s] an der Last/Slave *)
	lrAccMax							: LREAL;	(*maximale Beschleunigung [mm/s²] an der Last/Slave *)
	lrDecMax						: LREAL;	(*maximale Beschleunigung [mm/s²] an der Last/Slave *)

	i16_anzahl_mfps					: INT;
	lr_anfang_cam_table				: LREAL;
	lr_ende_cam_table				: LREAL;
END_VAR
VAR_OUTPUT
	bBusy							: BOOL;
	bDone							: BOOL;
	bError							: BOOL;
	udiErrorId						: UDINT;
	szErrText						: STRING;

	lrMasterVeloMax					: LREAL;
END_VAR
VAR
	stCamChar						: MC_TableCharacValues;	(*Charakteristika der Bewegungskurve*)
	fbReadCamTableCharacteristics	: MC_ReadCamTableCharacteristics;
	lrIncrement						: LREAL := 1;					(*Schrittweite Wertetabelle ACC / Integrationsschrittweite*)

	stVeloAccTable					: MC_CAM_Ref;
	aLrVeloAccData					: ARRAY[0..i_ANZAHL_PUNKTEMENGE,1..3] OF LREAL;	(*1..3  ->  MasterPos, SlaveVelo, SlaveAcc*)
	fbReadMotionFunctionValues		: MC_ReadMotionFunctionValues;
	(*===== INFO zu MotionFunktionValues: =====
	TYPE MC_ValueSelectType :
	(
	    (* a bitmask can be created by adding the following values *)
	    MC_VALUETYPE_POSITION     := 1,
	    MC_VALUETYPE_VELOCITY     := 2,
	    MC_VALUETYPE_ACCELERATION := 4,
	    MC_VALUETYPE_JERK         := 8
	);
	END_TYPE

	Mit der Auswahlmaske kann festgelegt werden, welche Daten interpoliert und zurückgeliefert werden soll.
	Der Wert entsteht durch Addition von Einzelwerten des Datentyps MC_ValueSelectType.
	Die Spaltenzahl der durch CamTable beschriebenen Datenstruktur muss der Anzahl der durch ValueSelectMask bestimmten Spaltenzahl entsprechen.
	Wenn zum Beispiel nur Positionsdaten gelesen werden, ist die Spaltenzahl 2 (Master- und Slave-Position).
	Mit jeder weiteren Ableitung (Geschwindigkeit, Beschleunigung, Ruck) kommt eine Spalte hinzu. *)

	lrMasterVelo1						: LREAL;	(*1.Mastergeschwindigkeit normiert aufgrund der max.Achsgeschwindigkeit*)
	lrMasterVelo2						: LREAL;	(*2.Reserve*)
	lrMasterVelo3						: LREAL;	(*3.Mastergeschwindigkeit normiert aufgrund der max.Achsbeschleunigung*)
	lrMasterVelo4						: LREAL;	(*4.Mastergeschwindigkeit normiert aufgrund der min.Achsbeschleunigung*)

	i								: INT;
	fb_state_entry						: ST_StateEntry;
END_VAR
VAR CONSTANT
	i_ANZAHL_PUNKTEMENGE		: INT := 360;
END_VAR
(* ======================================Schrittkette======================================== *)
fb_state_entry(
	i16_next_step:= ,
	i16_pos:= 1,
	s_debugtext:= ,
	E=> ,
	X=> ,
	i16_step=> ,
	i16_last_step=> );

CASE fb_state_entry.i16_step OF
(*=======================================================*)
	0 :	(* Init*)
		bBusy := FALSE;
		bDone := FALSE;
		bError := FALSE;
		udiErrorId := 0;
		szErrText := '';
		fbReadCamTableCharacteristics.Execute := FALSE;
		fbReadMotionFunctionValues.Execute := FALSE;
		fb_state_entry.i16_next_step := 10;

(*=======================================================*)
	10:	(* Warte Execute *)

		(*-----------------------Weiterschaltbedingungen----------------------------*)
		IF bExecute THEN
			bBusy := TRUE;
			fb_state_entry.i16_next_step := 20;
		END_IF

(*=======================================================*)
	20:	(* Prüfe Punktearray zur Anzeige der Punktewolke *)
		IF i16_anzahl_mfps > i_ANZAHL_PUNKTEMENGE THEN
			szErrText := 'Anzahl MFPs > Punktearray für Anzeige MF';
			fb_state_entry.i16_next_step := 1000;
		ELSE
			fb_state_entry.i16_next_step := 30;
		END_IF

(*=======================================================*)
	30:	(*Einlesen der Cam Table Characteristics*)
		IF fb_state_entry.E THEN
			fbReadCamTableCharacteristics.Execute := TRUE;
		END_IF

		(*-----------------------Weiterschaltbedingungen----------------------------*)
		IF fbReadCamTableCharacteristics.Busy THEN
			fb_state_entry.i16_next_step := 40;
		END_IF

(*=======================================================*)
	40:	(* Einlesen fertig  *)
		IF NOT fbReadCamTableCharacteristics.Busy THEN
			IF fbReadCamTableCharacteristics.Done THEN
				fbReadCamTableCharacteristics.Execute := FALSE;
				fb_state_entry.i16_next_step := 50;
			ELSIF fbReadCamTableCharacteristics.Error THEN
				udiErrorId := fbReadCamTableCharacteristics.ErrorID;
				szErrText := 'Fehler Einlesen charakteristische Daten';
				fb_state_entry.i16_next_step := 1000;
			END_IF
		END_IF

(*=======================================================*)
	50:	(*Geschwindigkeitsfunktion und Beschleunigungsfunktion lesen*)
		(*Upload der anzuzeigenden Punktewolke: masterPos, slaveVelo, slaveAcc mit MC_ReadMotionFunctionValues*)
		IF fb_state_entry.E THEN
			stVeloAccTable.ArraySize := SIZEOF(aLrVeloAccData);
			stVeloAccTable.pArray := ADR(aLrVeloAccData);
			stVeloAccTable.NoOfColumns := 3;	(*MasterPos, SlaveVelo, SlaveAcc*)
			stVeloAccTable.NoOfRows := i_ANZAHL_PUNKTEMENGE + 1;
			stVeloAccTable.TableType := MC_TABLETYPE_EQUIDISTANT;

			fbReadMotionFunctionValues.Execute := TRUE;
		END_IF

		(*-----------------------Weiterschaltbedingungen----------------------------*)
		IF fbReadMotionFunctionValues.Busy THEN
			fb_state_entry.i16_next_step := 60;
		END_IF

(*=======================================================*)
	60:	(* Einlesen fertig  *)
		IF NOT fbReadMotionFunctionValues.Busy THEN
			IF fbReadMotionFunctionValues.Done THEN
				fbReadMotionFunctionValues.Execute := FALSE;
				fb_state_entry.i16_next_step := 70;
			ELSIF fbReadMotionFunctionValues.Error THEN
				udiErrorId := fbReadMotionFunctionValues.ErrorID;
				szErrText := 'Beschleunigungsfunktion ungültig';
				fb_state_entry.i16_next_step := 1000;
			END_IF
		END_IF

(*=======================================================*)
	70:	(*  Berechnung der maximalen Mastergeschwindigkeit auf der Basis *)
		(*  der antriebsbedingten maximalen Geschwindigkeit des Slaves und der Tabelle.*)
		IF fb_state_entry.E THEN
			IF bEvCamTableChar THEN
				stCamChar.fSlaveVeloMin := 0;
				stCamChar.fSlaveVeloMax := 0;
				stCamChar.fSlaveAccMin := 0;
				stCamChar.fSlaveAccMax := 0;
				(* Ermittle Min- und Max-Werte für SlaveVelo und Slave Acc aus den interpolierten Daten in der Tabelle *)
				FOR i := 1 TO i_ANZAHL_PUNKTEMENGE DO
					IF aLrVeloAccData[i,2] > stCamChar.fSlaveVeloMax THEN
						stCamChar.fSlaveVeloMax := aLrVeloAccData[i,2];	(* an Position 2 -> SlaveVeloMax *)
					END_IF
					IF aLrVeloAccData[i,2] < stCamChar.fSlaveVeloMin THEN
						stCamChar.fSlaveVeloMin := aLrVeloAccData[i,2];	(* an Position 2 -> SlaveVeloMin *)
					END_IF
					IF aLrVeloAccData[i,3] > stCamChar.fSlaveAccMax THEN
						stCamChar.fSlaveAccMax := aLrVeloAccData[i,3];	(* an Position 3 -> SlaveAccMax *)
					END_IF
					IF aLrVeloAccData[i,3] < stCamChar.fSlaveAccMin THEN
						stCamChar.fSlaveAccMin := aLrVeloAccData[i,3];	(* an Position 3 -> SlaveAccMin *)
					END_IF
				END_FOR
			END_IF
		END_IF
		(*Fehlerbehandlung: Charakteristische Daten nicht konsistent*)
		(*Slave-Maximal- und Minimalgeschwindigkeit = 0*)
		IF stCamChar.fSlaveVeloMax = 0 AND stCamChar.fSlaveVeloMin = 0 THEN
			szErrText := 'Slave-Maximalgeschwindigkeit = 0';
			fb_state_entry.i16_next_step := 1000;
		(*Slave-Maximalbeschleunigung = 0*)
		ELSIF stCamChar.fSlaveAccMax = 0 THEN
			FOR i := 1 TO i_ANZAHL_PUNKTEMENGE DO
				IF aLrVeloAccData[i,3] > stCamChar.fSlaveAccMax THEN
					stCamChar.fSlaveAccMax := aLrVeloAccData[i,3];
				END_IF
			END_FOR
			IF stCamChar.fSlaveAccMax = 0 THEN
				szErrText := 'Slave-Maximalbeschleunigung = 0';
				fb_state_entry.i16_next_step := 1000;
			END_IF
		(*Slave-Minimalbeschleunigung = 0*)
		ELSIF stCamChar.fSlaveAccMin = 0 THEN
			FOR i := 1 TO i_ANZAHL_PUNKTEMENGE DO
				IF aLrVeloAccData[i,3] < stCamChar.fSlaveAccMin THEN
					stCamChar.fSlaveAccMin := aLrVeloAccData[i,3];
				END_IF
			END_FOR
			IF stCamChar.fSlaveAccMin = 0 THEN
				szErrText := 'Slave-Minimalbeschleunigung = 0';
				fb_state_entry.i16_next_step := 1000;
			END_IF
		(* Alles o.k. *)
		ELSE
			fb_state_entry.i16_next_step := 80;
		END_IF

	(*=======================================================*)
	80:	(*  Berechnung der maximalen Mastergeschwindigkeit  *)
		IF fb_state_entry.E THEN
			(* Im Kurvenscheibeneditor des Systemmanagers kann die "Normierte Darstellung" angehakt werden. *)
			(* Damit wird die Darstellung auf die maximale Achsgeschwindigkeit normiert. *)
			(*1.Mastergeschwindigkeit normiert aufgrund der max.Achsgeschwindigkeit*)
			(*Vs = Vm * Vf *)
			lrMasterVelo1 := ABS(lrVeloMax) / MAX(ABS(stCamChar.fSlaveVeloMin), ABS(stCamChar.fSlaveVeloMax));
			(*2.Reserve*)
			lrMasterVelo2 := lrMasterVelo1;
			(*3.Mastergeschwindigkeit normiert aufgrund der positiven Achsbeschleunigung*)
			(*As = Af(Sm)*Vm² + Vf(Sm)*Am *)
			lrMasterVelo3 := SQRT(ABS(MAX(lrAccMax,lrDecMax)) / ABS(stCamChar.fSlaveAccMax));
			(*4.Mastergeschwindigkeit normiert aufgrund der negativen Achsbeschleunigung*)
			(*As = Af(Sm)*Vm² + Vf(Sm)*Am *)
			lrMasterVelo4 := SQRT(ABS(MAX(lrAccMax,lrDecMax)) / ABS(stCamChar.fSlaveAccMin));
	
			lrMasterVeloMax := MIN(lrMasterVelo1, lrMasterVelo2);
			lrMasterVeloMax := MIN(lrMasterVeloMax, lrMasterVelo3);
			lrMasterVeloMax := MIN(lrMasterVeloMax, lrMasterVelo4);
		END_IF

		(*-----------------------Weiterschaltbedingungen----------------------------*)
		IF lrMasterVeloMax > 0 THEN
			fb_state_entry.i16_next_step := 90;
		ELSE
			szErrText := 'Master-Maximalbeschleunigung <= 0';
			fb_state_entry.i16_next_step := 1000;
		END_IF

(*=======================================================*)
	90: (* Fertig *)
		IF fb_state_entry.E THEN
			bBusy := FALSE;
			bDone := TRUE;
		END_IF

		(*-----------------------Weiterschaltbedingungen----------------------------*)
		IF NOT bExecute AND NOT fb_state_entry.E THEN
			 bDone := FALSE;
			fb_state_entry.i16_next_step := 10;
		END_IF

(*=======================================================*)
	1000: (* Fehler *)
		IF fb_state_entry.E THEN
			bError := TRUE;
			bBusy := FALSE;
		END_IF

		(*-----------------------Weiterschaltbedingungen----------------------------*)
		IF NOT bExecute THEN
			fb_state_entry.i16_next_step := 0;
		END_IF
END_CASE

fb_state_entry(
	i16_next_step:= ,
	i16_pos:= 2,
	s_debugtext:= ,
	E=> ,
	X=> ,
	i16_step=> ,
	i16_last_step=> );

fbReadCamTableCharacteristics(
	Execute:= ,
	CamTableID:=udiSlaveTableId,
	CamTableCharac:=stCamChar,
	Done=> ,
	Busy=> ,
	Error=> , 
	ErrorID=> );

fbReadMotionFunctionValues(
	Execute:= , 
	CamTableID:= udiSlaveTableId,
	ValueSelectMask:= MC_VALUETYPE_VELOCITY + MC_VALUETYPE_ACCELERATION,
	StartPosMaster:= lr_anfang_cam_table,
	EndPosMaster:= lr_ende_cam_table,
	Increment:= lrIncrement,
	CamTable:= stVeloAccTable,
	Done=> ,
	Busy=> , 
	Error=> ,
	ErrorID=> );
END_FUNCTION_BLOCK

(* POU EPT Lib/Funktionsbausteine/Nockenschaltwerke/NSW_INT/ST_Nockenschaltwerk_int, ST *)
FUNCTION_BLOCK ST_Nockenschaltwerk_int
VAR_INPUT
	i16_achsposition							: INT;
	i16_achsgeschwindigkeit					: INT;
	st_config									: struct_config;
END_VAR
VAR_IN_OUT
	st_visu									: struct_visu;
	arr_nocken								: ARRAY [0..15] OF struct_nocken_int;
END_VAR
VAR_OUTPUT
END_VAR
VAR
	b_first_cycle 								: BOOL := TRUE;
	i16_aktuelle_pos 							: INT := 0;
	i16_alte_pos	 							: INT := 0;
	r_zeit_fuer_1einheit						: REAL := 0.0;
	i16_anfangspos_mit_tzk 					: ARRAY [0..15] OF INT := 0;
	i16_endpos_mit_tzk 						: ARRAY [0..15] OF INT := 0;
	i16_vorsteuerpos_max						: INT := 0;
	b_verfahrrichtung_positiv 					: BOOL := FALSE;
	b_verfahrrichtung_negativ					: BOOL := FALSE;
	sm_positionseingabe						: BOOL := FALSE;
	sm_vorsteuerung							: BOOL := FALSE;
	sp, no									: UINT := 0;
	arr_spur									: ARRAY [0..15] OF BOOL;
	b_setzustand_anfang_kleiner_ende			: ARRAY [0..15] OF BOOL;
	b_setzustand_anfang_groesser_ende		: ARRAY [0..15] OF BOOL;
	b_resetzustand_anfang_kleiner_ende		: ARRAY [0..15] OF BOOL;
	b_resetzustand_anfang_groesser_ende		: ARRAY [0..15] OF BOOL;
END_VAR
(* Funktionsbaustein Nockenschaltwerk *)
IF b_first_cycle THEN
	b_first_cycle := FALSE;
	i16_vorsteuerpos_max := 60;
	b_verfahrrichtung_positiv := TRUE;
	b_verfahrrichtung_negativ := FALSE;
	i16_alte_pos := i16_aktuelle_pos;
END_IF

(* Aktuelle Position für weitere Komponenten zur Verfügung stellen *)
i16_aktuelle_pos := i16_achsposition;

(* Verfahrrichtung überwachen *)
IF i16_aktuelle_pos > i16_alte_pos THEN
	b_verfahrrichtung_positiv := TRUE;
	b_verfahrrichtung_negativ := FALSE;
	i16_alte_pos := i16_aktuelle_pos;
ELSIF i16_aktuelle_pos < i16_alte_pos THEN
	b_verfahrrichtung_positiv := FALSE;
	b_verfahrrichtung_negativ := TRUE;
	i16_alte_pos := i16_aktuelle_pos;
END_IF

IF i16_achsgeschwindigkeit >= 1 THEN
	(* 0.006 = 360Grad / (60sec * 1000ms) *)
	r_zeit_fuer_1einheit := 0.006 * INT_TO_REAL(i16_achsgeschwindigkeit);	(* REAL-Zahl in ms *)
ELSE
	r_zeit_fuer_1einheit := 0.0;
END_IF

(* Erst alle Spuren reset *)
FOR sp := 0  TO SIZEOF (arr_spur)/SIZEOF(arr_spur[0]) - 1BY 1 DO
	arr_spur[sp] :=FALSE;
END_FOR

(* Totzeitkompensation durch Vorsteuerung *)
FOR no := 0  TO SIZEOF (arr_nocken)/SIZEOF(arr_nocken[0]) - 1 BY 1DO
	(* Berechnung des Vorsteuerwinkels *)
	arr_nocken[no].i16_vorsteuerpos :=  REAL_TO_INT((TIME_TO_REAL(arr_nocken[no].t_vorsteuerzeit)) * r_zeit_fuer_1einheit);
	IF  arr_nocken[no].i16_vorsteuerpos >=i16_vorsteuerpos_max THEN
		 arr_nocken[no].i16_vorsteuerpos := 0;
		sm_vorsteuerung := TRUE;
	ELSE
		sm_vorsteuerung := FALSE;
	END_IF

	(* Nockentoleranz mit Berücksichtigung der Vorsteuerzeit für Anfangswinkel*)
	i16_anfangspos_mit_tzk[no] := arr_nocken[no].i16_cam_begin -  arr_nocken[no].i16_vorsteuerpos;
	IF i16_anfangspos_mit_tzk[no] > 360 THEN
		i16_anfangspos_mit_tzk[no] := i16_anfangspos_mit_tzk[no] - 360;
	ELSIF i16_anfangspos_mit_tzk[no] < 0 THEN
		i16_anfangspos_mit_tzk[no] := i16_anfangspos_mit_tzk[no] + 360;
	END_IF
	(* Nockentoleranz mit Berücksichtigung der Vorsteuerzeit für Endwinkel*)
	i16_endpos_mit_tzk[no] := arr_nocken[no].i16_cam_end -  arr_nocken[no].i16_vorsteuerpos;
	IF i16_endpos_mit_tzk[no] > 360 THEN
		i16_endpos_mit_tzk[no] := i16_endpos_mit_tzk[no] - 360;
	ELSIF i16_endpos_mit_tzk[no] < 0 THEN
		i16_endpos_mit_tzk[no] := i16_endpos_mit_tzk[no] + 360;
	END_IF

	IF i16_anfangspos_mit_tzk[no] < 0 OR i16_endpos_mit_tzk[no] < 0 OR i16_anfangspos_mit_tzk[no] >= 360 OR i16_endpos_mit_tzk[no] >= 360 THEN
		 (* Fehlerfälle  mit Abbruch*)
		sm_positionseingabe := TRUE;
		EXIT; (* Schleifenabbruch *)
	ELSE (* Winkel sind o.k. und der Nocken wird bearbeitet -> ON/OFF *)
		sm_positionseingabe := FALSE;
		IF i16_anfangspos_mit_tzk[no] <> i16_endpos_mit_tzk[no] THEN
			(* Nocken setzen *)
			(* Anfangswinkel ist kleiner Endwinkel *)
			b_setzustand_anfang_kleiner_ende[no] := i16_anfangspos_mit_tzk[no] < i16_endpos_mit_tzk[no] AND
												i16_aktuelle_pos >= i16_anfangspos_mit_tzk[no] AND
												i16_aktuelle_pos <= i16_endpos_mit_tzk[no];
			(* Anfangswinkel ist grösser Endwinkel *)
			b_setzustand_anfang_groesser_ende[no] := i16_anfangspos_mit_tzk[no] > i16_endpos_mit_tzk[no] AND
												(i16_aktuelle_pos >= i16_anfangspos_mit_tzk[no] OR
												i16_aktuelle_pos <= i16_endpos_mit_tzk[no]);

			(* Nocken ist gültig, d.h. wurde von der Maschine oder Bediener aktiviert *)
			IF	arr_nocken[no].b_camvalid AND
				(b_setzustand_anfang_kleiner_ende[no] OR b_setzustand_anfang_groesser_ende[no]) AND
				((b_verfahrrichtung_positiv AND arr_nocken[no].b_eff_direction_pos) OR	(* positive Drehrichtung und positive Wirkrichtung ist freigegeben *)
				(b_verfahrrichtung_negativ AND arr_nocken[no].b_eff_direction_neg)) 		(* negative Drehrichtung und negative Wirkrichtung ist freigegeben *)
				THEN
					arr_nocken[no].b_nockenzustand := TRUE;
			END_IF

			(* Nocken zurücksetzen *)
			(* Anfangswinkel ist kleiner Endwinkel *)
			b_resetzustand_anfang_kleiner_ende[no] := i16_anfangspos_mit_tzk[no] < i16_endpos_mit_tzk[no] AND
													(i16_aktuelle_pos < i16_anfangspos_mit_tzk[no] OR
													i16_aktuelle_pos  > i16_endpos_mit_tzk[no]);
			(* Anfangswinkel ist grösser Endwinkel *)
			b_resetzustand_anfang_groesser_ende[no] := i16_anfangspos_mit_tzk[no] > i16_endpos_mit_tzk[no] AND
													i16_aktuelle_pos < i16_anfangspos_mit_tzk[no] AND
													i16_aktuelle_pos > i16_endpos_mit_tzk[no];

			(* Nocken ist ungültig, d.h. wurde von der Maschine oder Bediener deaktiviert *)
			IF	NOT arr_nocken[no].b_camvalid OR
				(b_resetzustand_anfang_kleiner_ende[no] OR b_resetzustand_anfang_groesser_ende[no])
				THEN
					arr_nocken[no].b_nockenzustand := FALSE;
			END_IF
		ELSE
			(* Anfang = Ende -> Nocken ist false *)
			arr_nocken[no].b_nockenzustand := FALSE;
		END_IF
	END_IF

	(* Aktive Nocken auf ihre Spuren setzen *)
	IF arr_nocken[no].b_camvalid AND arr_nocken[no].b_nockenzustand THEN
		arr_spur[arr_nocken[no].i16_track_no] := TRUE;
	END_IF
END_FOR

IF st_config.b_config_fertig THEN
	(* Fehlermeldungen und Betriebsmeldungen ab dem Startindex in die globalen Meldungsarrays schreiben *)
	garr_stoermeldungen[st_config.i16_meld_startindex + 0] := sm_positionseingabe;
	garr_stoermeldungen[st_config.i16_meld_startindex + 1] := sm_vorsteuerung;
	garr_stoermeldungen[st_config.i16_meld_startindex + 2] := FALSE;
	garr_stoermeldungen[st_config.i16_meld_startindex + 3] := FALSE;
	garr_stoermeldungen[st_config.i16_meld_startindex + 4] := FALSE;
	garr_stoermeldungen[st_config.i16_meld_startindex + 5] := FALSE;
	garr_stoermeldungen[st_config.i16_meld_startindex + 6] := FALSE;
	garr_stoermeldungen[st_config.i16_meld_startindex + 7] := FALSE;
	garr_stoermeldungen[st_config.i16_meld_startindex + 8] := FALSE;
	garr_stoermeldungen[st_config.i16_meld_startindex + 9] := FALSE;
	garr_stoermeldungen[st_config.i16_meld_startindex + 10] := FALSE;
	garr_stoermeldungen[st_config.i16_meld_startindex + 11] := FALSE;
	garr_stoermeldungen[st_config.i16_meld_startindex + 12] := FALSE;
	garr_stoermeldungen[st_config.i16_meld_startindex + 13] := FALSE;
	garr_stoermeldungen[st_config.i16_meld_startindex + 14] := FALSE;
	garr_stoermeldungen[st_config.i16_meld_startindex + 15] := FALSE;
	garr_stoermeldungen[st_config.i16_meld_startindex + 16] := FALSE;
	garr_stoermeldungen[st_config.i16_meld_startindex + 17] := FALSE;
	garr_stoermeldungen[st_config.i16_meld_startindex + 18] := FALSE;
	garr_stoermeldungen[st_config.i16_meld_startindex + 19] := FALSE;
	
	garr_betriebsmeldungen[st_config.i16_meld_startindex + 0] := FALSE;
	garr_betriebsmeldungen[st_config.i16_meld_startindex + 1] := FALSE;
	garr_betriebsmeldungen[st_config.i16_meld_startindex + 2] := FALSE;
	garr_betriebsmeldungen[st_config.i16_meld_startindex + 3] := FALSE;
	garr_betriebsmeldungen[st_config.i16_meld_startindex + 4] := FALSE;
	garr_betriebsmeldungen[st_config.i16_meld_startindex + 5] := FALSE;
	garr_betriebsmeldungen[st_config.i16_meld_startindex + 6] := FALSE;
	garr_betriebsmeldungen[st_config.i16_meld_startindex + 7] := FALSE;
	garr_betriebsmeldungen[st_config.i16_meld_startindex + 8] := FALSE;
	garr_betriebsmeldungen[st_config.i16_meld_startindex + 9] := FALSE;
	garr_betriebsmeldungen[st_config.i16_meld_startindex + 10] := FALSE;
	garr_betriebsmeldungen[st_config.i16_meld_startindex + 11] := FALSE;
	garr_betriebsmeldungen[st_config.i16_meld_startindex + 12] := FALSE;
	garr_betriebsmeldungen[st_config.i16_meld_startindex + 13] := FALSE;
	garr_betriebsmeldungen[st_config.i16_meld_startindex + 14] := FALSE;
	garr_betriebsmeldungen[st_config.i16_meld_startindex + 15] := FALSE;
	garr_betriebsmeldungen[st_config.i16_meld_startindex + 16] := FALSE;
	garr_betriebsmeldungen[st_config.i16_meld_startindex + 17] := FALSE;
	garr_betriebsmeldungen[st_config.i16_meld_startindex + 18] := FALSE;
	garr_betriebsmeldungen[st_config.i16_meld_startindex + 19] := FALSE;
END_IF
END_FUNCTION_BLOCK

(* POU EPT Lib/Funktionsbausteine/Nockenschaltwerke/NSW_LREAL/ST_Nockenschaltwerk_lreal, ST *)
FUNCTION_BLOCK ST_Nockenschaltwerk_lreal
VAR_INPUT
	r_achsposition							: LREAL;
	r_achsgeschwindigkeit						: LREAL;
	i16_verfahrrichtung_achse_extern			: INT;
	b_verfahrrichtungsauswertung_extern			: BOOL;
	i16_art_der_achse							: enum_ecd_typ;
	st_config									: struct_config;
END_VAR
VAR_IN_OUT
	st_visu									: struct_visu;
	arr_nocken								: ARRAY [0..MAX_NOCKENGERUEST] OF struct_nocken_lreal;
END_VAR
VAR_OUTPUT
END_VAR
VAR
	b_first_cycle 								: BOOL := TRUE;
	r_aktuelle_pos 							: T_FIX16;
	r_alte_pos	 							: T_FIX16;
	b_verfahrrichtung_positiv 					: BOOL := FALSE;
	b_verfahrrichtung_negativ					: BOOL := FALSE;
	r_zeit_fuer_1einheit						: LREAL := 0.0;
	r_anfangspos_mit_tzk 						: ARRAY [0..MAX_NOCKENGERUEST] OF LREAL := 0.0;
	r_endpos_mit_tzk 							: ARRAY [0..MAX_NOCKENGERUEST] OF LREAL := 0.0;
	r_vorsteuerpos_max						: LREAL := 0.0;
	i16_verfahrrichtung_achse_intern				: INT := 0;
	sm_positionseingabe						: BOOL := FALSE;
	sm_vorsteuerung							: BOOL := FALSE;
	sp, no									: UINT := 0;
	arr_spur									: ARRAY [0..MAX_NOCKENGERUEST] OF BOOL;
	b_setzustand_anfang_kleiner_ende			: ARRAY [0..MAX_NOCKENGERUEST] OF BOOL;
	b_setzustand_anfang_groesser_ende		: ARRAY [0..MAX_NOCKENGERUEST] OF BOOL;
	b_resetzustand_anfang_kleiner_ende		: ARRAY [0..MAX_NOCKENGERUEST] OF BOOL;
	b_resetzustand_anfang_groesser_ende		: ARRAY [0..MAX_NOCKENGERUEST] OF BOOL;
END_VAR
(* Funktionsbaustein Nockenschaltwerk *)
(* Funktion für lineare und rotatorische Achsen *)
CASE i16_art_der_achse  OF
1:	(* Linearachse *)
	IF b_first_cycle THEN
		b_first_cycle := FALSE;

		(* Setze Drehrichtung Positiv. Da wenn beide Drehrichtungen nicht gesetzt sind, keine Nocke aktiv wird *)
		r_vorsteuerpos_max := 100.0;
		b_verfahrrichtung_positiv := TRUE;
		b_verfahrrichtung_negativ := FALSE;
		r_alte_pos := r_aktuelle_pos;
	END_IF

	(* Aktuelle Position für weitere Komponenten zur Verfügung stellen *)
	r_aktuelle_pos := LREAL_TO_FIX16(r_achsposition,2);

	(* Verfahrrichtung überwachen *)
	IF FIX16_TO_LREAL(r_aktuelle_pos) > FIX16_TO_LREAL(r_alte_pos) THEN
		i16_verfahrrichtung_achse_intern := 1;
		r_alte_pos := r_aktuelle_pos;
	ELSIF FIX16_TO_LREAL(r_aktuelle_pos) < FIX16_TO_LREAL(r_alte_pos) THEN
		i16_verfahrrichtung_achse_intern := -1;
		r_alte_pos := r_aktuelle_pos;
	END_IF

	IF b_verfahrrichtungsauswertung_extern THEN
		IF i16_verfahrrichtung_achse_extern = 1 THEN
			b_verfahrrichtung_positiv := TRUE;
			b_verfahrrichtung_negativ := FALSE;
		ELSIF i16_verfahrrichtung_achse_extern = -1 THEN
			b_verfahrrichtung_positiv := FALSE;
			b_verfahrrichtung_negativ := TRUE;
		END_IF
	ELSE
		IF i16_verfahrrichtung_achse_intern = 1 THEN
			b_verfahrrichtung_positiv := TRUE;
			b_verfahrrichtung_negativ := FALSE;
		ELSIF i16_verfahrrichtung_achse_intern = -1 THEN
			b_verfahrrichtung_positiv := FALSE;
			b_verfahrrichtung_negativ := TRUE;
		END_IF
	END_IF

	IF r_achsgeschwindigkeit >= 1.0 THEN
		r_zeit_fuer_1einheit := 0.001 * r_achsgeschwindigkeit;		(* REAL-Zahl in ms *)
	ELSE
		r_zeit_fuer_1einheit := 0.0;
	END_IF

	(* Totzeitkompensation durch Vorsteuerung *)
	FOR no := 0  TO SIZEOF (arr_nocken)/SIZEOF(arr_nocken[0]) -1 DO
		(* Berechnung der Vorsteuerposition *)
		 arr_nocken[no].r_vorsteuerpos :=  (TIME_TO_LREAL(arr_nocken[no].t_vorsteuerzeit)) * r_zeit_fuer_1einheit;
		IF  arr_nocken[no].r_vorsteuerpos >= r_vorsteuerpos_max THEN
			 arr_nocken[no].r_vorsteuerpos := 0.0;
			sm_vorsteuerung := TRUE;
		ELSE
			sm_vorsteuerung := FALSE;
		END_IF

		(* Nockentoleranz mit Berücksichtigung der Vorsteuerzeit für Anfangswinkel*)
		r_anfangspos_mit_tzk[no] := arr_nocken[no].r_cam_begin - arr_nocken[no].r_vorsteuerpos;
		(* Nockentoleranz mit Berücksichtigung der Vorsteuerzeit für Endwinkel*)
		r_endpos_mit_tzk[no] := arr_nocken[no].r_cam_end - arr_nocken[no].r_vorsteuerpos;

		IF r_anfangspos_mit_tzk[no] <> r_endpos_mit_tzk[no] THEN
			(* Nocken setzen *)
			(* Anfangsposition ist kleiner Endposition *)
			b_setzustand_anfang_kleiner_ende[no] := r_anfangspos_mit_tzk[no] < r_endpos_mit_tzk[no] AND
													FIX16_TO_LREAL(r_aktuelle_pos) >= r_anfangspos_mit_tzk[no] AND
													FIX16_TO_LREAL(r_aktuelle_pos) <= r_endpos_mit_tzk[no];
			(* Anfangsposition ist grösser Endposition *)
			b_setzustand_anfang_groesser_ende[no] := r_anfangspos_mit_tzk[no] > r_endpos_mit_tzk[no] AND
													FIX16_TO_LREAL(r_aktuelle_pos) <= r_anfangspos_mit_tzk[no] AND
													FIX16_TO_LREAL(r_aktuelle_pos) >= r_endpos_mit_tzk[no];
	
			(* Nocken ist gültig, d.h. wurde von der Maschine oder Bediener aktiviert *)
			IF	arr_nocken[no].b_camvalid AND
				(b_setzustand_anfang_kleiner_ende[no] OR b_setzustand_anfang_groesser_ende[no]) AND
				((b_verfahrrichtung_positiv AND arr_nocken[no].b_eff_direction_pos) OR	(* positive Drehrichtung und positive Wirkrichtung ist freigegeben *)
				(b_verfahrrichtung_negativ AND arr_nocken[no].b_eff_direction_neg)) 		(* negative Drehrichtung und negative Wirkrichtung ist freigegeben *)
				THEN
					arr_nocken[no].b_nockenzustand := TRUE;
			END_IF
	
			(* Nocken zurücksetzen *)
			(* Anfangswinkel ist kleiner Endwinkel *)
			b_resetzustand_anfang_kleiner_ende[no] := r_anfangspos_mit_tzk[no] < r_endpos_mit_tzk[no] AND
													(FIX16_TO_LREAL(r_aktuelle_pos) < r_anfangspos_mit_tzk[no] OR
													FIX16_TO_LREAL(r_aktuelle_pos)  > r_endpos_mit_tzk[no]);
			(* Anfangswinkel ist grösser Endwinkel *)
			b_resetzustand_anfang_groesser_ende[no] := r_anfangspos_mit_tzk[no] > r_endpos_mit_tzk[no] AND
													(FIX16_TO_LREAL(r_aktuelle_pos) > r_anfangspos_mit_tzk[no] OR
													FIX16_TO_LREAL(r_aktuelle_pos) < r_endpos_mit_tzk[no]);
	
			(* Nocken ist ungültig, d.h. wurde von der Maschine oder Bediener deaktiviert *)
			IF	NOT arr_nocken[no].b_camvalid OR
				b_resetzustand_anfang_kleiner_ende[no] OR
				b_resetzustand_anfang_groesser_ende[no] OR
				(* Zusatzbedingung für Nockenzustand rücksetzen ist nur bei Linearachsen sinnvoll *)
				(b_verfahrrichtung_positiv AND NOT arr_nocken[no].b_eff_direction_pos AND arr_nocken[no].b_eff_direction_neg) OR	(* positive Drehrichtung und positive Wirkrichtung ist freigegeben *)
				(b_verfahrrichtung_negativ AND NOT arr_nocken[no].b_eff_direction_neg AND arr_nocken[no].b_eff_direction_pos)		(* negative Drehrichtung und negative Wirkrichtung ist freigegeben *)
				THEN
					arr_nocken[no].b_nockenzustand := FALSE;
			END_IF
		ELSE
			(* Anfang = Ende -> Nocken ist false *)
			arr_nocken[no].b_nockenzustand := FALSE;
		END_IF
	END_FOR

	(* Erst alle Spuren reset *)
	FOR sp := 0  TO SIZEOF (arr_spur)-1 DO
		arr_spur[sp] :=FALSE;
	END_FOR
	
	(* Dann aktive Nocken auf ihre Spuren setzen *)
	FOR no := 0  TO SIZEOF (arr_nocken)/SIZEOF(arr_nocken[0])-1 DO
		IF arr_nocken[no].b_camvalid AND arr_nocken[no].b_nockenzustand THEN
			arr_spur[arr_nocken[no].i16_track_no] := TRUE;
		END_IF
	END_FOR

2:	(* Rotatorische Achse *)
	IF b_first_cycle THEN
		b_first_cycle := FALSE;

		(* Setze Drehrichtung Positiv. Da wenn beide Drehrichtungen nicht gesetzt sind, keine Nocke aktiv wird *)
		r_vorsteuerpos_max := 60.0;
		b_verfahrrichtung_positiv := TRUE;
		b_verfahrrichtung_negativ := FALSE;
		r_alte_pos := r_aktuelle_pos;
	END_IF

	(* Aktuelle Position für weitere Komponenten zur Verfügung stellen *)
	r_aktuelle_pos := LREAL_TO_FIX16(r_achsposition,2);

	(* Verfahrrichtung überwachen *)
	IF FIX16_TO_LREAL(r_aktuelle_pos) > FIX16_TO_LREAL(r_alte_pos) THEN
		i16_verfahrrichtung_achse_intern := 1;
		r_alte_pos := r_aktuelle_pos;
	ELSIF FIX16_TO_LREAL(r_aktuelle_pos) < FIX16_TO_LREAL(r_alte_pos) THEN
		i16_verfahrrichtung_achse_intern := -1;
		r_alte_pos := r_aktuelle_pos;
	END_IF

	IF b_verfahrrichtungsauswertung_extern THEN
		IF i16_verfahrrichtung_achse_extern = 1 THEN
			b_verfahrrichtung_positiv := TRUE;
			b_verfahrrichtung_negativ := FALSE;
		ELSIF i16_verfahrrichtung_achse_extern = -1 THEN
			b_verfahrrichtung_positiv := FALSE;
			b_verfahrrichtung_negativ := TRUE;
		END_IF
	ELSE
		IF i16_verfahrrichtung_achse_intern = 1 THEN
			b_verfahrrichtung_positiv := TRUE;
			b_verfahrrichtung_negativ := FALSE;
		ELSIF i16_verfahrrichtung_achse_intern = -1 THEN
			b_verfahrrichtung_positiv := FALSE;
			b_verfahrrichtung_negativ := TRUE;
		END_IF
	END_IF

	IF r_achsgeschwindigkeit >= 1.0 THEN
		(* 0.006 = 360Grad / (60sec * 1000ms) *)
		r_zeit_fuer_1einheit := 0.006 * r_achsgeschwindigkeit;	(* REAL-Zahl in ms *)
	ELSE
		r_zeit_fuer_1einheit := 0.0;
	END_IF

	(* Totzeitkompensation durch Vorsteuerung *)
	FOR no := 0  TO SIZEOF (arr_nocken)/SIZEOF(arr_nocken[0]) -1 DO
		(* Berechnung des Vorsteuerwinkels *)
		arr_nocken[no].r_vorsteuerpos :=  (TIME_TO_LREAL(arr_nocken[no].t_vorsteuerzeit)) * r_zeit_fuer_1einheit;
		IF  arr_nocken[no].r_vorsteuerpos >= r_vorsteuerpos_max THEN
			 arr_nocken[no].r_vorsteuerpos := 0.0;
			sm_vorsteuerung := TRUE;
		ELSE
			sm_vorsteuerung := FALSE;
		END_IF

		(* Nockentoleranz mit Berücksichtigung der Vorsteuerzeit für Anfangswinkel*)
		r_anfangspos_mit_tzk[no] := arr_nocken[no].r_cam_begin -  arr_nocken[no].r_vorsteuerpos;
		IF r_anfangspos_mit_tzk[no] > 360.0 THEN
			r_anfangspos_mit_tzk[no] := r_anfangspos_mit_tzk[no] - 360.0;
		ELSIF r_anfangspos_mit_tzk[no] < 0.0 THEN
			r_anfangspos_mit_tzk[no] := r_anfangspos_mit_tzk[no] + 360.0;
		END_IF
		(* Nockentoleranz mit Berücksichtigung der Vorsteuerzeit für Endwinkel*)
		r_endpos_mit_tzk[no] := arr_nocken[no].r_cam_end -  arr_nocken[no].r_vorsteuerpos;
		IF r_endpos_mit_tzk[no] > 360.0 THEN
			r_endpos_mit_tzk[no] := r_endpos_mit_tzk[no] - 360.0;
		ELSIF r_endpos_mit_tzk[no] < 0.0 THEN
			r_endpos_mit_tzk[no] := r_endpos_mit_tzk[no] + 360.0;
		END_IF
	
		IF r_anfangspos_mit_tzk[no] < 0.0 OR r_endpos_mit_tzk[no] < 0.0 OR r_anfangspos_mit_tzk[no] >= 360.0 OR r_endpos_mit_tzk[no] >= 360.0 THEN
			 (* Fehlerfälle  mit Abbruch*)
			sm_positionseingabe := TRUE;
			EXIT; (* Schleifenabbruch *)
		ELSE (* Winkel sind o.k. und der Nocken wird bearbeitet -> ON/OFF *)
			sm_positionseingabe := FALSE;
			IF r_anfangspos_mit_tzk[no] <> r_endpos_mit_tzk[no] THEN
				(* Nocken setzen *)
				(* Anfangswinkel ist kleiner Endwinkel *)
				b_setzustand_anfang_kleiner_ende[no] := r_anfangspos_mit_tzk[no] < r_endpos_mit_tzk[no] AND
													FIX16_TO_LREAL(r_aktuelle_pos) >= r_anfangspos_mit_tzk[no] AND
													FIX16_TO_LREAL(r_aktuelle_pos) <= r_endpos_mit_tzk[no];
				(* Anfangswinkel ist grösser Endwinkel *)
				b_setzustand_anfang_groesser_ende[no] := r_anfangspos_mit_tzk[no] > r_endpos_mit_tzk[no] AND
													(FIX16_TO_LREAL(r_aktuelle_pos) >= r_anfangspos_mit_tzk[no] OR
													FIX16_TO_LREAL(r_aktuelle_pos) <= r_endpos_mit_tzk[no]);

				(* Nocken ist gültig, d.h. wurde von der Maschine oder Bediener aktiviert *)
				IF	arr_nocken[no].b_camvalid AND
					(b_setzustand_anfang_kleiner_ende[no] OR b_setzustand_anfang_groesser_ende[no]) AND
					((b_verfahrrichtung_positiv AND arr_nocken[no].b_eff_direction_pos) OR	(* positive Drehrichtung und positive Wirkrichtung ist freigegeben *)
					(b_verfahrrichtung_negativ AND arr_nocken[no].b_eff_direction_neg)) 		(* negative Drehrichtung und negative Wirkrichtung ist freigegeben *)
					THEN
						arr_nocken[no].b_nockenzustand := TRUE;
				END_IF

				(* Nocken zurücksetzen *)
				(* Anfangswinkel ist kleiner Endwinkel *)
				b_resetzustand_anfang_kleiner_ende[no] := r_anfangspos_mit_tzk[no] < r_endpos_mit_tzk[no] AND
														(FIX16_TO_LREAL(r_aktuelle_pos) < r_anfangspos_mit_tzk[no] OR
														FIX16_TO_LREAL(r_aktuelle_pos)  > r_endpos_mit_tzk[no]);
				(* Anfangswinkel ist grösser Endwinkel *)
				b_resetzustand_anfang_groesser_ende[no] := r_anfangspos_mit_tzk[no] > r_endpos_mit_tzk[no] AND
														FIX16_TO_LREAL(r_aktuelle_pos) < r_anfangspos_mit_tzk[no] AND
														FIX16_TO_LREAL(r_aktuelle_pos) > r_endpos_mit_tzk[no];

				(* Nocken ist ungültig, d.h. wurde von der Maschine oder Bediener deaktiviert *)
				IF	NOT arr_nocken[no].b_camvalid OR
					(b_resetzustand_anfang_kleiner_ende[no] OR b_resetzustand_anfang_groesser_ende[no])
					THEN
						arr_nocken[no].b_nockenzustand := FALSE;
				END_IF
			ELSE
				(* Anfang = Ende -> Nocken ist false *)
				arr_nocken[no].b_nockenzustand := FALSE;
			END_IF
		END_IF
	END_FOR

	(* Erst alle Spuren reset *)
	FOR sp := 0  TO SIZEOF (arr_spur)-1 DO
		arr_spur[sp] :=FALSE;
	END_FOR

	(* Dann aktive Nocken auf ihre Spuren setzen *)
	FOR no := 0  TO SIZEOF (arr_nocken)/SIZEOF(arr_nocken[0])-1 DO
		IF arr_nocken[no].b_camvalid AND arr_nocken[no].b_nockenzustand THEN
			arr_spur[arr_nocken[no].i16_track_no] := TRUE;
		END_IF
	END_FOR
END_CASE

IF st_config.b_config_fertig THEN
	(* Fehlermeldungen und Betriebsmeldungen ab dem Startindex in die globalen Meldungsarrays schreiben *)
	garr_stoermeldungen[st_config.i16_meld_startindex + 0] := sm_positionseingabe;
	garr_stoermeldungen[st_config.i16_meld_startindex + 1] := sm_vorsteuerung;
	garr_stoermeldungen[st_config.i16_meld_startindex + 2] := FALSE;
	garr_stoermeldungen[st_config.i16_meld_startindex + 3] := FALSE;
	garr_stoermeldungen[st_config.i16_meld_startindex + 4] := FALSE;
	garr_stoermeldungen[st_config.i16_meld_startindex + 5] := FALSE;
	garr_stoermeldungen[st_config.i16_meld_startindex + 6] := FALSE;
	garr_stoermeldungen[st_config.i16_meld_startindex + 7] := FALSE;
	garr_stoermeldungen[st_config.i16_meld_startindex + 8] := FALSE;
	garr_stoermeldungen[st_config.i16_meld_startindex + 9] := FALSE;
	garr_stoermeldungen[st_config.i16_meld_startindex + 10] := FALSE;
	garr_stoermeldungen[st_config.i16_meld_startindex + 11] := FALSE;
	garr_stoermeldungen[st_config.i16_meld_startindex + 12] := FALSE;
	garr_stoermeldungen[st_config.i16_meld_startindex + 13] := FALSE;
	garr_stoermeldungen[st_config.i16_meld_startindex + 14] := FALSE;
	garr_stoermeldungen[st_config.i16_meld_startindex + 15] := FALSE;
	garr_stoermeldungen[st_config.i16_meld_startindex + 16] := FALSE;
	garr_stoermeldungen[st_config.i16_meld_startindex + 17] := FALSE;
	garr_stoermeldungen[st_config.i16_meld_startindex + 18] := FALSE;
	garr_stoermeldungen[st_config.i16_meld_startindex + 19] := FALSE;
	
	garr_betriebsmeldungen[st_config.i16_meld_startindex + 0] := FALSE;
	garr_betriebsmeldungen[st_config.i16_meld_startindex + 1] := FALSE;
	garr_betriebsmeldungen[st_config.i16_meld_startindex + 2] := FALSE;
	garr_betriebsmeldungen[st_config.i16_meld_startindex + 3] := FALSE;
	garr_betriebsmeldungen[st_config.i16_meld_startindex + 4] := FALSE;
	garr_betriebsmeldungen[st_config.i16_meld_startindex + 5] := FALSE;
	garr_betriebsmeldungen[st_config.i16_meld_startindex + 6] := FALSE;
	garr_betriebsmeldungen[st_config.i16_meld_startindex + 7] := FALSE;
	garr_betriebsmeldungen[st_config.i16_meld_startindex + 8] := FALSE;
	garr_betriebsmeldungen[st_config.i16_meld_startindex + 9] := FALSE;
	garr_betriebsmeldungen[st_config.i16_meld_startindex + 10] := FALSE;
	garr_betriebsmeldungen[st_config.i16_meld_startindex + 11] := FALSE;
	garr_betriebsmeldungen[st_config.i16_meld_startindex + 12] := FALSE;
	garr_betriebsmeldungen[st_config.i16_meld_startindex + 13] := FALSE;
	garr_betriebsmeldungen[st_config.i16_meld_startindex + 14] := FALSE;
	garr_betriebsmeldungen[st_config.i16_meld_startindex + 15] := FALSE;
	garr_betriebsmeldungen[st_config.i16_meld_startindex + 16] := FALSE;
	garr_betriebsmeldungen[st_config.i16_meld_startindex + 17] := FALSE;
	garr_betriebsmeldungen[st_config.i16_meld_startindex + 18] := FALSE;
	garr_betriebsmeldungen[st_config.i16_meld_startindex + 19] := FALSE;
END_IF
END_FUNCTION_BLOCK

(* POU EPT Lib/Funktionsbausteine/Nockenschaltwerke/NZW/ST_Nockenzaehlwerk, ST *)
FUNCTION_BLOCK ST_Nockenzaehlwerk
VAR_INPUT
	i16_wkz_vorbesetzwert		: INT;
	b_zustand_spur			: BOOL;
	b_externer_zaehler_reset	: BOOL;
END_VAR
VAR_OUTPUT
	b_aktionsnocken			: BOOL;
END_VAR
VAR
	fb_ctu_hubzaehler			: CTU;
	fb_r_trig_zaehler			: R_TRIG;
	fb_r_trig_ot_nocken		: R_TRIG;
	b_interner_zaehler_reset	: BOOL := FALSE;
END_VAR
(* Zählwerk für Aktionen, die OT-Nocken abhängig sind
Anwendung: Nacheiner bestimmten Anzahl von Umdrehungen soll eine Aktion ausgelöst werden.
Der Ausgang ist für eine Umdrehung aktiv, bevor er wieder zurückgesetzt wird. *)
fb_ctu_hubzaehler(
	CU:=  b_zustand_spur,
	RESET:= b_interner_zaehler_reset OR b_externer_zaehler_reset,
	PV:= i16_wkz_vorbesetzwert,
	Q=> ,
	CV=> );

fb_r_trig_zaehler(CLK:= fb_ctu_hubzaehler.Q, Q=> );

(* Abfrage des Zählerstatus und daraus resultierende Aktionen *)
IF fb_r_trig_zaehler.Q THEN (* Bei Zählerstand erreicht, Ausgang für eine Umdrehung setzen *)
	b_aktionsnocken := TRUE;
END_IF
IF NOT fb_ctu_hubzaehler.Q AND fb_r_trig_ot_nocken.Q THEN
	b_aktionsnocken := FALSE; (* Nach einer Umdrehung wird der Ausgang wieder rückgesetzt *)
END_IF

fb_r_trig_ot_nocken(CLK:= b_zustand_spur, Q=> );

IF NOT  b_zustand_spur AND fb_ctu_hubzaehler.Q THEN
	b_interner_zaehler_reset := TRUE; (* Wenn Zählerstand erreicht, dann Zähler nullen *)
ELSIF b_interner_zaehler_reset AND fb_ctu_hubzaehler.CV = 0 THEN
	b_interner_zaehler_reset := FALSE; (* Wenn Zähler genullt, dann wieder freigeben für erneutes Zählen *)
END_IF
END_FUNCTION_BLOCK

(* POU EPT Lib/Programmbausteine/ST_Start_Batchscript, ST *)
FUNCTION_BLOCK ST_Start_Batchscript
VAR_INPUT
	bExecute			: BOOL;
	bQuit				: BOOL;
	st_pfad				: STRING;
END_VAR
VAR_OUTPUT
	bBusy				: BOOL;
	bReady				: BOOL;
	bError				: BOOL;
	nErrId				: UDINT;
END_VAR
VAR
	fb_ton_quitt					: TON;
	fb_state_entry					: ST_StateEntry;
	fb_r_trig_execute				: R_TRIG;
	fb_nt_start_process			: NT_StartProcess;
END_VAR
(* Starten eines Batchscriptes auf dem lokalen PC *)
fb_r_trig_execute(CLK:= bExecute, Q=> );
fb_ton_quitt(IN:= , PT:= t#100ms, Q=> , ET=> );

fb_state_entry(
	i16_next_step:= ,
	i16_pos:= 1,
	s_debugtext:= ,
	E=> ,
	X=> , 
	i16_step=> ,
	i16_last_step=> );

CASE fb_state_entry.i16_step OF
(*=======================================================*)
	0:(* INIT *)
		bBusy := FALSE;
		bReady := FALSE;
		bError := FALSE;
		nErrId := 0;
		fb_nt_start_process.START := FALSE;
		fb_state_entry.i16_next_step := 10;

(*=======================================================*)
	10:	(* Warte auf Execute-Befehl *)

		IF fb_r_trig_execute.Q THEN
			bReady := FALSE;
			bBusy := TRUE;
			fb_state_entry.i16_next_step := 20;
		END_IF

(*=======================================================*)
	20:	(* Starte mit Ausführen des Batchscriptes *)
		IF fb_state_entry.E THEN
			fb_nt_start_process.START := TRUE;
		END_IF

		IF fb_nt_start_process.BUSY THEN
			fb_nt_start_process.START := FALSE;
			fb_state_entry.i16_next_step := 30;
		END_IF

(*=======================================================*)
	30:	(* Script wurde erfolgreich ausgeführt *)
		IF NOT fb_nt_start_process.BUSY THEN
			IF NOT fb_nt_start_process.ERR THEN
				bBusy := FALSE;
				fb_state_entry.i16_next_step := 999;
			ELSE	(* Fehler *)
				fb_state_entry.i16_next_step := 1000;
			END_IF
		END_IF

(*=======================================================*)
	999:	(* Fertig *)
		bReady := TRUE;
		fb_state_entry.i16_next_step := 10;

(*=======================================================*)
	1000: (* Fehler *)
		IF fb_state_entry.E THEN
			bBusy := FALSE;
			bReady := FALSE;
			bError := TRUE;
			fb_ton_quitt.IN := FALSE;
		END_IF

		(*-----------------------Weiterschaltbedingungen----------------------------*)
		IF bQuit AND NOT fb_state_entry.E THEN
			bError := FALSE;
			fb_ton_quitt.IN := TRUE;
		END_IF

		IF fb_ton_quitt.Q THEN
			fb_ton_quitt.IN := FALSE;
			fb_state_entry.i16_next_step := 0;
		END_IF
END_CASE

fb_state_entry(
	i16_next_step:= , 
	i16_pos:= 2,
	s_debugtext:= ,
	E=> ,
	X=> ,
	i16_step=> ,
	i16_last_step=> );

fb_nt_start_process(
	NETID:= '',
	PATHSTR:= st_pfad,
	DIRNAME:= , 
	COMNDLINE:= ,
	START:= ,
	TMOUT:= DEFAULT_ADS_TIMEOUT,
	BUSY=> ,
	ERR=> , 
	ERRID=> nErrId);
END_FUNCTION_BLOCK

(* POU Gemeinsamkeiten17xx/Stueckzahlen/ST_Stueckzahl, ST *)
FUNCTION_BLOCK ST_Stueckzahl
VAR_INPUT
	b_wkz_zweifachfallend			: BOOL;
	st_config						: struct_config;
	st_ctrl_in						: struct_ctrl_in;
END_VAR
VAR_OUTPUT
	st_ctrl_out					: struct_ctrl_out;
END_VAR
VAR
	fb_ton_wz					: TON;
	fb_ton_uez					: TON;
	fb_ton_quitt					: TON;
	fb_r_trig_gutteil				: R_TRIG;
	fb_r_trig_schlechtteil			: R_TRIG;
	fb_state_entry					: ST_StateEntry;
	i							: INT;
	sm_auftrag_voll				: BOOL := FALSE;
	sm_verpackungseinheit_voll	: BOOL := FALSE;
	i16_faktor_wkz				: INT := 1;
END_VAR
(* Zeiten *)
fb_ton_wz(IN:= , PT:= , Q=>  , ET=> );
fb_ton_uez(IN:= , PT:= , Q=>  , ET=> );
fb_ton_quitt(IN:= , PT:= t#100ms, Q=> , ET=> );

(* Flanken *)
fb_r_trig_gutteil(CLK:= st_ctrl_in.b_gutteil_produziert, Q=> );
fb_r_trig_schlechtteil(CLK:= st_ctrl_in.b_schlechtteil_produziert, Q=> );


IF b_wkz_zweifachfallend THEN
	i16_faktor_wkz := 2;
ELSE
	i16_faktor_wkz := 1;
END_IF

(* Toplevel *)
IF fb_state_entry.i16_next_step > INIT AND fb_state_entry.i16_next_step < FEHLER THEN
	IF fb_state_entry.i16_next_step < STOP THEN
		IF st_ctrl_in.b_stop THEN
			fb_state_entry.i16_next_step := STOP;
		END_IF
	END_IF

	(* Zählerstände rücksetzen *)
	FOR i := 0 TO (SIZEOF (gst_datensatz.st_stueckzahlen.st_teilezaehler) / SIZEOF (gst_datensatz.st_stueckzahlen.st_teilezaehler[0])) - 1  BY 1 DO
		IF gst_datensatz.st_stueckzahlen.st_teilezaehler[i].b_reset_gutteile THEN
			gst_datensatz.st_stueckzahlen.st_teilezaehler[i].i32_aktuelle_gutteile := 0;
		END_IF
		IF gst_datensatz.st_stueckzahlen.st_teilezaehler[i].b_reset_schlechtteile THEN
			gst_datensatz.st_stueckzahlen.st_teilezaehler[i].i32_aktuelle_schlechtteile := 0;
		END_IF
	END_FOR
END_IF

(* ==================================Schrittkette================================ *)
fb_state_entry(
	i16_next_step:= , 
	i16_pos:= 1,
	s_debugtext:= ,
	E=> ,
	X=> , 
	i16_step=> ,
	i16_last_step=> );

CASE fb_state_entry.i16_step OF
(*=======================================================*)
	INIT_OBJ:
		IF st_config.b_config_fertig THEN
			fb_state_entry.i16_next_step := INIT;
		END_IF

(*=======================================================*)
	INIT:
		IF fb_state_entry.E THEN
			fb_ton_wz.IN := FALSE;
			fb_ton_uez.IN := FALSE;
			fb_ton_quitt.IN := FALSE;
			sm_auftrag_voll := FALSE;
			sm_verpackungseinheit_voll := FALSE;
			st_ctrl_out.b_fehler := FALSE;
			st_ctrl_out.b_bereit := FALSE;
			st_ctrl_out.b_fertig := FALSE;
		END_IF

		(*-----------------------Weiterschaltbedingungen----------------------------*)
		IF st_ctrl_in.b_init THEN
			fb_state_entry.i16_next_step := BEREIT;
		END_IF

(*=======================================================*)
	BEREIT:
		IF fb_state_entry.E THEN
			st_ctrl_out.b_bereit := TRUE;
		END_IF

		(* Zähler hochzählen *)
		IF fb_r_trig_gutteil.Q THEN
			gst_datensatz.st_stueckzahlen.st_teilezaehler[JAHR].i32_aktuelle_gutteile := gst_datensatz.st_stueckzahlen.st_teilezaehler[JAHR].i32_aktuelle_gutteile + i16_faktor_wkz;
			gst_datensatz.st_stueckzahlen.st_teilezaehler[VPE].i32_aktuelle_gutteile := gst_datensatz.st_stueckzahlen.st_teilezaehler[VPE].i32_aktuelle_gutteile + i16_faktor_wkz;
		END_IF

		IF fb_r_trig_schlechtteil.Q THEN
			gst_datensatz.st_stueckzahlen.st_teilezaehler[JAHR].i32_aktuelle_schlechtteile := gst_datensatz.st_stueckzahlen.st_teilezaehler[JAHR].i32_aktuelle_schlechtteile + i16_faktor_wkz;
			gst_datensatz.st_stueckzahlen.st_teilezaehler[VPE].i32_aktuelle_schlechtteile := gst_datensatz.st_stueckzahlen.st_teilezaehler[VPE].i32_aktuelle_schlechtteile + i16_faktor_wkz;
		END_IF

		(* Eine Verpackungseinheit ist voll *)
		IF 	gst_datensatz.st_stueckzahlen.st_teilezaehler[VPE].i32_aktuelle_gutteile >= gst_datensatz.st_stueckzahlen.st_teilezaehler[VPE].i32_vorgabe_gutteile AND
			fb_state_entry.i16_next_step <> FEHLER
			THEN
				gst_datensatz.st_stueckzahlen.st_teilezaehler[AUFTRAG].i32_aktuelle_gutteile := gst_datensatz.st_stueckzahlen.st_teilezaehler[AUFTRAG].i32_aktuelle_gutteile + 1;
				sm_verpackungseinheit_voll := TRUE;
				fb_state_entry.i16_next_step := FEHLER;
		END_IF
		(* Gesamter Auftrag ist voll *)
		IF 	gst_datensatz.st_stueckzahlen.st_teilezaehler[AUFTRAG].i32_aktuelle_gutteile >= gst_datensatz.st_stueckzahlen.st_teilezaehler[AUFTRAG].i32_vorgabe_gutteile AND
			fb_state_entry.i16_next_step <> FEHLER
			THEN
				sm_auftrag_voll := TRUE;
				fb_state_entry.i16_next_step := FEHLER;
		END_IF

(*=======================================================*)
	FEHLER:
		IF fb_state_entry.E THEN
			st_ctrl_out.b_fehler := TRUE;
		END_IF

		(*-----------------------Weiterschaltbedingungen----------------------------*)
		IF st_ctrl_in.b_quitt AND NOT fb_state_entry.E THEN
			st_ctrl_out.b_fehler := FALSE;
			fb_ton_quitt.IN := TRUE;

			IF gst_datensatz.st_stueckzahlen.st_teilezaehler[VPE].i32_aktuelle_gutteile >= gst_datensatz.st_stueckzahlen.st_teilezaehler[VPE].i32_vorgabe_gutteile THEN
				gst_datensatz.st_stueckzahlen.st_teilezaehler[VPE].i32_aktuelle_gutteile := 0;
				sm_verpackungseinheit_voll := FALSE;
			END_IF
			IF gst_datensatz.st_stueckzahlen.st_teilezaehler[AUFTRAG].i32_aktuelle_gutteile >= gst_datensatz.st_stueckzahlen.st_teilezaehler[AUFTRAG].i32_vorgabe_gutteile THEN
				gst_datensatz.st_stueckzahlen.st_teilezaehler[AUFTRAG].i32_aktuelle_gutteile := 0;
				sm_auftrag_voll := FALSE;
			END_IF
		END_IF

		IF fb_ton_quitt.Q THEN
			fb_ton_quitt.IN := FALSE;
			fb_state_entry.i16_next_step := INIT;
		END_IF

(*=======================================================*)
	STOP:

		(*-----------------------Weiterschaltbedingungen----------------------------*)
		IF st_ctrl_in.b_quitt AND NOT fb_state_entry.E THEN
			fb_ton_quitt.IN := TRUE;
		END_IF

		IF fb_ton_quitt.Q THEN
			fb_ton_quitt.IN := FALSE;
			fb_state_entry.i16_next_step := INIT;
		END_IF
END_CASE

fb_state_entry(
	i16_next_step:= , 
	i16_pos:= 2,
	s_debugtext:= ,
	E=> , 
	X=> , 
	i16_step=> ,
	i16_last_step=> );

IF st_config.b_config_fertig THEN
	(* Fehlermeldungen und Betriebsmeldungen ab dem Startindex in die globalen Meldungsarrays schreiben *)
	garr_stoermeldungen[st_config.i16_meld_startindex + 0] := sm_verpackungseinheit_voll;
	garr_stoermeldungen[st_config.i16_meld_startindex + 1] := sm_auftrag_voll;
	garr_stoermeldungen[st_config.i16_meld_startindex + 2] := FALSE;
	garr_stoermeldungen[st_config.i16_meld_startindex + 3] := FALSE;
	garr_stoermeldungen[st_config.i16_meld_startindex + 4] := FALSE;
	garr_stoermeldungen[st_config.i16_meld_startindex + 5] := FALSE;
	garr_stoermeldungen[st_config.i16_meld_startindex + 6] := FALSE;
	garr_stoermeldungen[st_config.i16_meld_startindex + 7] := FALSE;
	garr_stoermeldungen[st_config.i16_meld_startindex + 8] := FALSE;
	garr_stoermeldungen[st_config.i16_meld_startindex + 9] := FALSE;
	garr_stoermeldungen[st_config.i16_meld_startindex + 10] := FALSE;
	garr_stoermeldungen[st_config.i16_meld_startindex + 11] := FALSE;
	garr_stoermeldungen[st_config.i16_meld_startindex + 12] := FALSE;
	garr_stoermeldungen[st_config.i16_meld_startindex + 13] := FALSE;
	garr_stoermeldungen[st_config.i16_meld_startindex + 14] := FALSE;
	garr_stoermeldungen[st_config.i16_meld_startindex + 15] := FALSE;
	garr_stoermeldungen[st_config.i16_meld_startindex + 16] := FALSE;
	garr_stoermeldungen[st_config.i16_meld_startindex + 17] := FALSE;
	garr_stoermeldungen[st_config.i16_meld_startindex + 18] := FALSE;
	garr_stoermeldungen[st_config.i16_meld_startindex + 19] := FALSE;
	
	garr_betriebsmeldungen[st_config.i16_meld_startindex + 0] := FALSE;
	garr_betriebsmeldungen[st_config.i16_meld_startindex + 1] := FALSE;
	garr_betriebsmeldungen[st_config.i16_meld_startindex + 2] := FALSE;
	garr_betriebsmeldungen[st_config.i16_meld_startindex + 3] := FALSE;
	garr_betriebsmeldungen[st_config.i16_meld_startindex + 4] := FALSE;
	garr_betriebsmeldungen[st_config.i16_meld_startindex + 5] := FALSE;
	garr_betriebsmeldungen[st_config.i16_meld_startindex + 6] := FALSE;
	garr_betriebsmeldungen[st_config.i16_meld_startindex + 7] := FALSE;
	garr_betriebsmeldungen[st_config.i16_meld_startindex + 8] := FALSE;
	garr_betriebsmeldungen[st_config.i16_meld_startindex + 9] := FALSE;
	garr_betriebsmeldungen[st_config.i16_meld_startindex + 10] := FALSE;
	garr_betriebsmeldungen[st_config.i16_meld_startindex + 11] := FALSE;
	garr_betriebsmeldungen[st_config.i16_meld_startindex + 12] := FALSE;
	garr_betriebsmeldungen[st_config.i16_meld_startindex + 13] := FALSE;
	garr_betriebsmeldungen[st_config.i16_meld_startindex + 14] := FALSE;
	garr_betriebsmeldungen[st_config.i16_meld_startindex + 15] := FALSE;
	garr_betriebsmeldungen[st_config.i16_meld_startindex + 16] := FALSE;
	garr_betriebsmeldungen[st_config.i16_meld_startindex + 17] := FALSE;
	garr_betriebsmeldungen[st_config.i16_meld_startindex + 18] := FALSE;
	garr_betriebsmeldungen[st_config.i16_meld_startindex + 19] := FALSE;
END_IF
END_FUNCTION_BLOCK

(* POU EPT Lib/Zylinder/ST_Zylinder12V012346E, ST *)
FUNCTION_BLOCK ST_Zylinder12V012346E
VAR_INPUT
	st_config							: struct_zylinder_config;
	bw_nocken_zylinder_einfahren		: BOOL;
	bw_nocken_zylinder_ausfahren		: BOOL;
	uw_nocken_zylinder_einfahren		: BOOL;
	uw_nocken_zylinder_ausfahren		: BOOL;
	b_direkttaste_ausfahren			: BOOL;
	b_direkttaste_mittefahren			: BOOL;
	b_direkttaste_einfahren				: BOOL;
	st_ctrl_in							: struct_zylinder_ctrl_in;
	e_druckwaechter					: BOOL;
	i16_betriebsart					: enum_betriebsarten;
	b_no_gesteuert_im_norm_betrieb	: BOOL;
	b_masterachse_hand_dialog_aktiv	: BOOL;
END_VAR
VAR_IN_OUT
	st_visu							: struct_zylinder_visu;
END_VAR
VAR_OUTPUT
	st_ctrl_out						: struct_zylinder_ctrl_out;
	a_ventil_einfahren					AT %Q* : BOOL;
	a_ventil_ausfahren				AT %Q* : BOOL;
END_VAR
VAR
	b_first_cycle 						: BOOL := TRUE;
	i16_anzahl_sensoren				: INT := 0;
	i16_anzahl_spulen					: INT := 0;
	b_sensor_eingefahren_vorhanden	: BOOL := FALSE;
	b_sensor_ausgefahren_vorhanden	: BOOL := FALSE;
	b_mit_tzk							: BOOL := FALSE;
	b_nockengesteuert				: BOOL := FALSE;
	b_zustand_uw_nocken_einfahren	: BOOL := FALSE;
	b_zustand_uw_nocken_ausfahren	: BOOL := FALSE;
	st_tzk							: struct_totzeitkompensation;
	fb_ton_uz_fahren					: TON;
	fb_ton_uz_endlage1				: TON;
	fb_ton_uz_endlage2				: TON;
	fb_ton_uz_endlage3				: TON;
	fb_ton_uz_sensor1					: TON;
	fb_ton_uz_sensor2					: TON;
	fb_ton_uz_sensor3					: TON;
	fb_ton_einausfahren				: TON;
	fb_r_trig_ibn_ausfahren				: R_TRIG;
	fb_r_trig_ibn_einfahren				: R_TRIG;
	fb_r_trig_ibn_quit					: R_TRIG;
	fb_ton_ibn_ausfahren				: TON;
	fb_ton_ibn_einfahren				: TON;
	fb_ton_ibn_quit					: TON;
	fb_ton_quitt						: TON;
	st_sm							: struct_zylinder_meldungen;
	fb_state_entry						: ST_StateEntry;
	b_ibn_zylinder_ausfahren			: BOOL := FALSE;
	b_ibn_zylinder_einfahren			: BOOL := FALSE;
	b_ibn_zylinderfehler_quit			: BOOL := FALSE;

	e_sensor1_eingefahren			AT %I* : BOOL;
	e_sensor1_ausgefahren			AT %I* : BOOL;
	e_sensor2_eingefahren			AT %I* : BOOL;
	e_sensor2_ausgefahren			AT %I* : BOOL;
	e_sensor3_eingefahren			AT %I* : BOOL;
	e_sensor3_ausgefahren			AT %I* : BOOL;
	e_sensor_mittegefahren			AT %I* : BOOL;
	e_taste_einfahren					AT %I* : BOOL;
	e_taste_ausfahren					AT %I* : BOOL;
END_VAR
IF b_first_cycle THEN
	b_first_cycle := FALSE;
	st_ctrl_out.b_fehler := FALSE;
	st_ctrl_out.b_eingefahren := FALSE;
	st_ctrl_out.b_ausgefahren := FALSE;
	st_ctrl_out.b_gestoppt := FALSE;
	st_sm.b_zeit_ausfahren1:= FALSE;
	st_sm.b_zeit_einfahren1:= FALSE;
	st_sm.b_endlage1	:= FALSE;
	st_sm.b_sensor1:= FALSE;
	st_sm.b_zeit_ausfahren2 := FALSE;
	st_sm.b_zeit_einfahren2 := FALSE;
	st_sm.b_endlage2	:= FALSE;
	st_sm.b_sensor2 := FALSE;
	st_sm.b_zeit_ausfahren3 := FALSE;
	st_sm.b_zeit_einfahren3 := FALSE;
	st_sm.b_endlage3	:= FALSE;
	st_sm.b_sensor3 := FALSE;
	st_sm.b_winkel_ausfahren1:= FALSE;
	st_sm.b_winkel_einfahren1:= FALSE;
	st_sm.b_winkel_ausfahren2 := FALSE;
	st_sm.b_winkel_einfahren2 := FALSE;
	st_sm.b_winkel_ausfahren3 := FALSE;
	st_sm.b_winkel_einfahren3 := FALSE;
	st_sm.b_zyltyp_nicht_definiert := FALSE;
	st_sm.b_reserve1:= FALSE;
END_IF

(* Inbetriebnahme *)
fb_r_trig_ibn_ausfahren(CLK:= b_ibn_zylinder_ausfahren, Q=> );
fb_r_trig_ibn_einfahren(CLK:= b_ibn_zylinder_einfahren, Q=> );
fb_r_trig_ibn_quit(CLK:= b_ibn_zylinderfehler_quit, Q=> );
fb_ton_ibn_ausfahren(IN:= , PT:= t#1s, Q=> , ET=> );
fb_ton_ibn_einfahren(IN:= , PT:= t#1s, Q=> , ET=> );
fb_ton_ibn_quit(IN:= , PT:= t#1s, Q=> , ET=> );
fb_ton_quitt(IN:= , PT:= t#50ms, Q=> , ET=> );

IF fb_r_trig_ibn_ausfahren.Q THEN
	fb_ton_ibn_ausfahren.IN := TRUE;
ELSE
	IF fb_ton_ibn_ausfahren.Q THEN
		b_ibn_zylinder_ausfahren := FALSE;
	 	fb_ton_ibn_ausfahren.IN := FALSE;
	END_IF
END_IF

IF fb_r_trig_ibn_einfahren.Q THEN
	fb_ton_ibn_einfahren.IN := TRUE;
ELSE
	IF fb_ton_ibn_einfahren.Q THEN
		b_ibn_zylinder_einfahren := FALSE;
	 	fb_ton_ibn_einfahren.IN := FALSE;
	END_IF
END_IF

IF fb_r_trig_ibn_quit.Q THEN
	fb_ton_ibn_quit.IN := TRUE;
ELSE
	IF fb_ton_ibn_quit.Q THEN
		b_ibn_zylinderfehler_quit := FALSE;
	 	fb_ton_ibn_quit.IN := FALSE;
	END_IF
END_IF

(* Simulationssensoren für den Zylinderhandbetrieb *)
IF  	gi16_betriebsart = HAND AND
	st_visu.i16_nr_zyl_im_handbetrieb = st_config.i16_identnummer AND
	fb_state_entry.i16_step > INIT_OBJ
	THEN
		CASE i16_anzahl_sensoren OF
			0:
				st_visu.b_sensor_mittegefahren := e_sensor_mittegefahren;
				st_visu.enu_zustand := fb_state_entry.i16_step;
			1:
				st_visu.b_sensor_ausgefahren := e_sensor1_ausgefahren;
				st_visu.b_sensor_eingefahren := e_sensor1_eingefahren;
				st_visu.enu_zustand := fb_state_entry.i16_step;
			2:
				IF b_sensor_eingefahren_vorhanden AND b_sensor_ausgefahren_vorhanden THEN
					st_visu.b_sensor_ausgefahren := e_sensor1_ausgefahren;
					st_visu.b_sensor_eingefahren := e_sensor1_eingefahren;
					st_visu.b_sensor_mittegefahren := e_sensor_mittegefahren;
				ELSIF b_sensor_ausgefahren_vorhanden THEN
					st_visu.b_sensor_ausgefahren := e_sensor1_ausgefahren OR e_sensor2_ausgefahren;
				ELSIF b_sensor_eingefahren_vorhanden THEN
					st_visu.b_sensor_eingefahren := e_sensor1_eingefahren OR e_sensor2_eingefahren;
				END_IF
				st_visu.enu_zustand := fb_state_entry.i16_step;
			4:
				st_visu.b_sensor_ausgefahren := e_sensor1_ausgefahren AND e_sensor2_ausgefahren;
				st_visu.b_sensor_eingefahren := e_sensor1_eingefahren AND e_sensor2_eingefahren;
				st_visu.b_sensor_mittegefahren := e_sensor_mittegefahren;
				st_visu.enu_zustand := fb_state_entry.i16_step;
			6:
				st_visu.b_sensor_ausgefahren := e_sensor1_ausgefahren AND e_sensor2_ausgefahren AND e_sensor3_ausgefahren;
				st_visu.b_sensor_eingefahren := e_sensor1_eingefahren AND e_sensor2_eingefahren AND e_sensor3_eingefahren;
				st_visu.b_sensor_mittegefahren := e_sensor_mittegefahren;
				st_visu.enu_zustand := fb_state_entry.i16_step;
		END_CASE
END_IF

(* Überwachungszeiten *)
fb_ton_uz_fahren(IN:= , PT:= st_config.t_ueberwachungszeit, Q=>  , ET=> );
fb_ton_uz_endlage1(IN:= , PT:= t#100ms, Q=> , ET=> );
fb_ton_uz_endlage2(IN:= , PT:= t#100ms, Q=> , ET=> );
fb_ton_uz_endlage3(IN:= , PT:= t#100ms, Q=> , ET=> );
fb_ton_uz_sensor1(IN:= , PT:= t#100ms, Q=> , ET=> );
fb_ton_uz_sensor2(IN:= , PT:= t#100ms, Q=> , ET=> );
fb_ton_uz_sensor3(IN:= , PT:= t#100ms, Q=> , ET=> );

(* Aus- und Einfahrzeit *)
fb_ton_einausfahren(IN:= , PT:= st_config.t_ein_aus_fahrzeit, Q=> , ET=> );

(* Totzeitkompensationszeit *)
st_tzk.fb_ton_tzk(IN:= , PT:= st_tzk.t_kompensationszeit, Q=> , ET=> );

IF fb_state_entry.i16_step > ZYL_INIT AND fb_state_entry.i16_step < ZYL_FEHLER THEN
	IF 	st_ctrl_in.b_stop AND
		(st_visu.i16_nr_zyl_im_handbetrieb <> st_config.i16_identnummer OR gi16_betriebsart <> HAND)
		THEN
			fb_state_entry.i16_next_step := GESTOPPT;
	END_IF
END_IF

(* Zylinder bewegen über Direkttasten von der hinteren Bedienoberfläche und Hardwaretaster *)
IF (b_direkttaste_ausfahren AND NOT b_direkttaste_einfahren) OR (e_taste_ausfahren AND NOT e_taste_einfahren) THEN
	fb_state_entry.i16_next_step := DIREKT_AUSFAHREN;
ELSIF (b_direkttaste_einfahren AND NOT b_direkttaste_ausfahren) OR (NOT e_taste_ausfahren AND e_taste_einfahren) THEN
	fb_state_entry.i16_next_step := DIREKT_EINFAHREN;
END_IF

(* ==================================Schrittkette================================ *)
fb_state_entry(
	i16_next_step:= ,
	i16_pos:= 1,
	s_debugtext:= ,
	E=> ,
	X=> ,
	i16_step=> ,
	i16_last_step=> );

